//     Term 38 (AT2200-0500)/CC Inputs/Current actual value Ch.30 <-> Data Pointer/CurrentActualValues[29]
//     Term 38 (AT2200-0500)/CC Inputs/Current actual value Ch.4 <-> Data Pointer/CurrentActualValues[3]
//     Term 38 (AT2200-0500)/CC Inputs/Current actual value Ch.5 <-> Data Pointer/CurrentActualValues[4]
//     Term 38 (AT2200-0500)/CC Inputs/Current actual value Ch.6 <-> Data Pointer/CurrentActualValues[5]
//     Term 38 (AT2200-0500)/CC Inputs/Current actual value Ch.7 <-> Data Pointer/CurrentActualValues[6]
//     Term 38 (AT2200-0500)/CC Inputs/Current actual value Ch.8 <-> Data Pointer/CurrentActualValues[7]
//     Term 38 (AT2200-0500)/CC Inputs/Current actual value Ch.9 <-> Data Pointer/CurrentActualValues[8]
//     Term 38 (AT2200-0500)/CC Inputs/Status <-> Data Pointer/Status
//     Term 38 (AT2200-0500)/CC Outputs/Control <-> Data Pointer/Control
//     Term 38 (AT2200-0500)/CC Outputs/Current setpoint value Ch.1 <-> Data Pointer/CurrentSetpointValues[0]
//     Term 38 (AT2200-0500)/CC Outputs/Current setpoint value Ch.10 <-> Data Pointer/CurrentSetpointValues[9]
//     Term 38 (AT2200-0500)/CC Outputs/Current setpoint value Ch.11 <-> Data Pointer/CurrentSetpointValues[10]
//     Term 38 (AT2200-0500)/CC Outputs/Current setpoint value Ch.12 <-> Data Pointer/CurrentSetpointValues[11]
//     Term 38 (AT2200-0500)/CC Outputs/Current setpoint value Ch.13 <-> Data Pointer/CurrentSetpointValues[12]
//     Term 38 (AT2200-0500)/CC Outputs/Current setpoint value Ch.14 <-> Data Pointer/CurrentSetpointValues[13]
//     Term 38 (AT2200-0500)/CC Outputs/Current setpoint value Ch.15 <-> Data Pointer/CurrentSetpointValues[14]
//     Term 38 (AT2200-0500)/CC Outputs/Current setpoint value Ch.16 <-> Data Pointer/CurrentSetpointValues[15]
//     Term 38 (AT2200-0500)/CC Outputs/Current setpoint value Ch.17 <-> Data Pointer/CurrentSetpointValues[16]
//     Term 38 (AT2200-0500)/CC Outputs/Current setpoint value Ch.18 <-> Data Pointer/CurrentSetpointValues[17]
//     Term 38 (AT2200-0500)/CC Outputs/Current setpoint value Ch.19 <-> Data Pointer/CurrentSetpointValues[18]
//     Term 38 (AT2200-0500)/CC Outputs/Current setpoint value Ch.2 <-> Data Pointer/CurrentSetpointValues[1]
//     Term 38 (AT2200-0500)/CC Outputs/Current setpoint value Ch.20 <-> Data Pointer/CurrentSetpointValues[19]
//     Term 38 (AT2200-0500)/CC Outputs/Current setpoint value Ch.21 <-> Data Pointer/CurrentSetpointValues[20]
//     Term 38 (AT2200-0500)/CC Outputs/Current setpoint value Ch.22 <-> Data Pointer/CurrentSetpointValues[21]
//     Term 38 (AT2200-0500)/CC Outputs/Current setpoint value Ch.23 <-> Data Pointer/CurrentSetpointValues[22]
//     Term 38 (AT2200-0500)/CC Outputs/Current setpoint value Ch.24 <-> Data Pointer/CurrentSetpointValues[23]
//     Term 38 (AT2200-0500)/CC Outputs/Current setpoint value Ch.25 <-> Data Pointer/CurrentSetpointValues[24]
//     Term 38 (AT2200-0500)/CC Outputs/Current setpoint value Ch.26 <-> Data Pointer/CurrentSetpointValues[25]
//     Term 38 (AT2200-0500)/CC Outputs/Current setpoint value Ch.27 <-> Data Pointer/CurrentSetpointValues[26]
//     Term 38 (AT2200-0500)/CC Outputs/Current setpoint value Ch.28 <-> Data Pointer/CurrentSetpointValues[27]
//     Term 38 (AT2200-0500)/CC Outputs/Current setpoint value Ch.29 <-> Data Pointer/CurrentSetpointValues[28]
//     Term 38 (AT2200-0500)/CC Outputs/Current setpoint value Ch.3 <-> Data Pointer/CurrentSetpointValues[2]
//     Term 38 (AT2200-0500)/CC Outputs/Current setpoint value Ch.30 <-> Data Pointer/CurrentSetpointValues[29]
//     Term 38 (AT2200-0500)/CC Outputs/Current setpoint value Ch.4 <-> Data Pointer/CurrentSetpointValues[3]
//     Term 38 (AT2200-0500)/CC Outputs/Current setpoint value Ch.5 <-> Data Pointer/CurrentSetpointValues[4]
//     Term 38 (AT2200-0500)/CC Outputs/Current setpoint value Ch.6 <-> Data Pointer/CurrentSetpointValues[5]
//     Term 38 (AT2200-0500)/CC Outputs/Current setpoint value Ch.7 <-> Data Pointer/CurrentSetpointValues[6]
//     Term 38 (AT2200-0500)/CC Outputs/Current setpoint value Ch.8 <-> Data Pointer/CurrentSetpointValues[7]
//     Term 38 (AT2200-0500)/CC Outputs/Current setpoint value Ch.9 <-> Data Pointer/CurrentSetpointValues[8]
//     Term 38 (AT2200-0500)/LFB Inputs/BinaryData <-> Data Pointer/HallSensorValues
//   Device 25 <-> TcCOM Objects/XTS ProcessingUnit 1/Part 1/Module 31
//     Term 39 (AT2000-0250)/CC Inputs/Current actual value Ch.1 <-> Data Pointer/CurrentActualValues[0]
//     Term 39 (AT2000-0250)/CC Inputs/Current actual value Ch.10 <-> Data Pointer/CurrentActualValues[9]
//     Term 39 (AT2000-0250)/CC Inputs/Current actual value Ch.11 <-> Data Pointer/CurrentActualValues[10]
//     Term 39 (AT2000-0250)/CC Inputs/Current actual value Ch.12 <-> Data Pointer/CurrentActualValues[11]
//     Term 39 (AT2000-0250)/CC Inputs/Current actual value Ch.13 <-> Data Pointer/CurrentActualValues[12]
//     Term 39 (AT2000-0250)/CC Inputs/Current actual value Ch.14 <-> Data Pointer/CurrentActualValues[13]
//     Term 39 (AT2000-0250)/CC Inputs/Current actual value Ch.15 <-> Data Pointer/CurrentActualValues[14]
//     Term 39 (AT2000-0250)/CC Inputs/Current actual value Ch.2 <-> Data Pointer/CurrentActualValues[1]
//     Term 39 (AT2000-0250)/CC Inputs/Current actual value Ch.3 <-> Data Pointer/CurrentActualValues[2]
//     Term 39 (AT2000-0250)/CC Inputs/Current actual value Ch.4 <-> Data Pointer/CurrentActualValues[3]
//     Term 39 (AT2000-0250)/CC Inputs/Current actual value Ch.5 <-> Data Pointer/CurrentActualValues[4]
//     Term 39 (AT2000-0250)/CC Inputs/Current actual value Ch.6 <-> Data Pointer/CurrentActualValues[5]
//     Term 39 (AT2000-0250)/CC Inputs/Current actual value Ch.7 <-> Data Pointer/CurrentActualValues[6]
//     Term 39 (AT2000-0250)/CC Inputs/Current actual value Ch.8 <-> Data Pointer/CurrentActualValues[7]
//     Term 39 (AT2000-0250)/CC Inputs/Current actual value Ch.9 <-> Data Pointer/CurrentActualValues[8]
//     Term 39 (AT2000-0250)/CC Inputs/Status <-> Data Pointer/Status
//     Term 39 (AT2000-0250)/CC Outputs/Control <-> Data Pointer/Control
//     Term 39 (AT2000-0250)/CC Outputs/Current setpoint value Ch.1 <-> Data Pointer/CurrentSetpointValues[0]
//     Term 39 (AT2000-0250)/CC Outputs/Current setpoint value Ch.10 <-> Data Pointer/CurrentSetpointValues[9]
//     Term 39 (AT2000-0250)/CC Outputs/Current setpoint value Ch.11 <-> Data Pointer/CurrentSetpointValues[10]
//     Term 39 (AT2000-0250)/CC Outputs/Current setpoint value Ch.12 <-> Data Pointer/CurrentSetpointValues[11]
//     Term 39 (AT2000-0250)/CC Outputs/Current setpoint value Ch.13 <-> Data Pointer/CurrentSetpointValues[12]
//     Term 39 (AT2000-0250)/CC Outputs/Current setpoint value Ch.14 <-> Data Pointer/CurrentSetpointValues[13]
//     Term 39 (AT2000-0250)/CC Outputs/Current setpoint value Ch.15 <-> Data Pointer/CurrentSetpointValues[14]
//     Term 39 (AT2000-0250)/CC Outputs/Current setpoint value Ch.2 <-> Data Pointer/CurrentSetpointValues[1]
//     Term 39 (AT2000-0250)/CC Outputs/Current setpoint value Ch.3 <-> Data Pointer/CurrentSetpointValues[2]
//     Term 39 (AT2000-0250)/CC Outputs/Current setpoint value Ch.4 <-> Data Pointer/CurrentSetpointValues[3]
//     Term 39 (AT2000-0250)/CC Outputs/Current setpoint value Ch.5 <-> Data Pointer/CurrentSetpointValues[4]
//     Term 39 (AT2000-0250)/CC Outputs/Current setpoint value Ch.6 <-> Data Pointer/CurrentSetpointValues[5]
//     Term 39 (AT2000-0250)/CC Outputs/Current setpoint value Ch.7 <-> Data Pointer/CurrentSetpointValues[6]
//     Term 39 (AT2000-0250)/CC Outputs/Current setpoint value Ch.8 <-> Data Pointer/CurrentSetpointValues[7]
//     Term 39 (AT2000-0250)/CC Outputs/Current setpoint value Ch.9 <-> Data Pointer/CurrentSetpointValues[8]
//     Term 39 (AT2000-0250)/Term 40 (AT2000-5250)/FB Inputs/Value Channel 01 <-> Data Pointer/RawPositionValues[0]
//     Term 39 (AT2000-0250)/Term 40 (AT2000-5250)/FB Inputs/Value Channel 02 <-> Data Pointer/RawPositionValues[1]
//     Term 39 (AT2000-0250)/Term 40 (AT2000-5250)/FB Inputs/Value Channel 03 <-> Data Pointer/RawPositionValues[2]
//     Term 39 (AT2000-0250)/Term 40 (AT2000-5250)/FB Inputs/Value Channel 04 <-> Data Pointer/RawPositionValues[3]
//     Term 39 (AT2000-0250)/Term 40 (AT2000-5250)/FB Inputs/Value Channel 05 <-> Data Pointer/RawPositionValues[4]
//     Term 39 (AT2000-0250)/Term 40 (AT2000-5250)/FB Inputs/Value Channel 06 <-> Data Pointer/RawPositionValues[5]
//     Term 39 (AT2000-0250)/Term 40 (AT2000-5250)/FB Inputs/Value Channel 07 <-> Data Pointer/RawPositionValues[6]
//     Term 39 (AT2000-0250)/Term 40 (AT2000-5250)/FB Inputs/Value Channel 08 <-> Data Pointer/RawPositionValues[7]
//     Term 39 (AT2000-0250)/Term 40 (AT2000-5250)/FB Inputs/Value Channel 09 <-> Data Pointer/RawPositionValues[8]
//     Term 39 (AT2000-0250)/Term 40 (AT2000-5250)/FB Inputs/Value Channel 10 <-> Data Pointer/RawPositionValues[9]
//     Term 39 (AT2000-0250)/Term 40 (AT2000-5250)/FB Inputs/Value Channel 11 <-> Data Pointer/RawPositionValues[10]
//     Term 39 (AT2000-0250)/Term 40 (AT2000-5250)/FB Inputs/Value Channel 12 <-> Data Pointer/RawPositionValues[11]
//     Term 39 (AT2000-0250)/Term 40 (AT2000-5250)/FB Inputs/Value Channel 13 <-> Data Pointer/RawPositionValues[12]
//     Term 39 (AT2000-0250)/Term 40 (AT2000-5250)/FB Inputs/Value Channel 14 <-> Data Pointer/RawPositionValues[13]
//     Term 39 (AT2000-0250)/Term 40 (AT2000-5250)/FB Inputs/Value Channel 15 <-> Data Pointer/RawPositionValues[14]
//     Term 39 (AT2000-0250)/Term 40 (AT2000-5250)/FB Inputs/Value Channel 16 <-> Data Pointer/RawPositionValues[15]
//     Term 39 (AT2000-0250)/Term 40 (AT2000-5250)/FB Inputs/Value Channel 17 <-> Data Pointer/RawPositionValues[16]
//     Term 39 (AT2000-0250)/Term 40 (AT2000-5250)/FB Inputs/Value Channel 18 <-> Data Pointer/RawPositionValues[17]
//     Term 39 (AT2000-0250)/Term 40 (AT2000-5250)/FB Inputs/Value Channel 19 <-> Data Pointer/RawPositionValues[18]
//     Term 39 (AT2000-0250)/Term 40 (AT2000-5250)/FB Inputs/Value Channel 20 <-> Data Pointer/RawPositionValues[19]
//     Term 39 (AT2000-0250)/Term 40 (AT2000-5250)/FB Inputs/Value Channel 21 <-> Data Pointer/RawPositionValues[20]
//     Term 39 (AT2000-0250)/Term 40 (AT2000-5250)/FB Inputs/Value Channel 22 <-> Data Pointer/RawPositionValues[21]
//     Term 39 (AT2000-0250)/Term 40 (AT2000-5250)/FB Inputs/Value Channel 23 <-> Data Pointer/RawPositionValues[22]
//     Term 39 (AT2000-0250)/Term 40 (AT2000-5250)/FB Inputs/Value Channel 24 <-> Data Pointer/RawPositionValues[23]
//     Term 39 (AT2000-0250)/Term 40 (AT2000-5250)/FB Inputs/Value Channel 25 <-> Data Pointer/RawPositionValues[24]
//     Term 39 (AT2000-0250)/Term 40 (AT2000-5250)/FB Inputs/Value Channel 26 <-> Data Pointer/RawPositionValues[25]
//     Term 39 (AT2000-0250)/Term 40 (AT2000-5250)/FB Inputs/Value Channel 27 <-> Data Pointer/RawPositionValues[26]
//     Term 39 (AT2000-0250)/Term 40 (AT2000-5250)/FB Inputs/Value Channel 28 <-> Data Pointer/RawPositionValues[27]
//     Term 39 (AT2000-0250)/Term 40 (AT2000-5250)/FB Inputs/Value Channel 29 <-> Data Pointer/RawPositionValues[28]
//     Term 39 (AT2000-0250)/Term 40 (AT2000-5250)/FB Inputs/Value Channel 30 <-> Data Pointer/RawPositionValues[29]
//     Term 39 (AT2000-0250)/Term 40 (AT2000-5250)/FB Inputs/Value Channel 31 <-> Data Pointer/RawPositionValues[30]
//     Term 39 (AT2000-0250)/Term 40 (AT2000-5250)/FB Inputs/Value Channel 32 <-> Data Pointer/RawPositionValues[31]
//   Device 26 <-> TcCOM Objects/XTS ProcessingUnit 1/Part 1/Module 32
//     Term 41 (AT2002-0250)/CC Inputs/Current actual value Ch.1 <-> Data Pointer/CurrentActualValues[0]
//     Term 41 (AT2002-0250)/CC Inputs/Current actual value Ch.10 <-> Data Pointer/CurrentActualValues[9]
//     Term 41 (AT2002-0250)/CC Inputs/Current actual value Ch.11 <-> Data Pointer/CurrentActualValues[10]
//     Term 41 (AT2002-0250)/CC Inputs/Current actual value Ch.12 <-> Data Pointer/CurrentActualValues[11]
//     Term 41 (AT2002-0250)/CC Inputs/Current actual value Ch.13 <-> Data Pointer/CurrentActualValues[12]
//     Term 41 (AT2002-0250)/CC Inputs/Current actual value Ch.14 <-> Data Pointer/CurrentActualValues[13]
//     Term 41 (AT2002-0250)/CC Inputs/Current actual value Ch.15 <-> Data Pointer/CurrentActualValues[14]
//     Term 41 (AT2002-0250)/CC Inputs/Current actual value Ch.2 <-> Data Pointer/CurrentActualValues[1]
//     Term 41 (AT2002-0250)/CC Inputs/Current actual value Ch.3 <-> Data Pointer/CurrentActualValues[2]
//     Term 41 (AT2002-0250)/CC Inputs/Current actual value Ch.4 <-> Data Pointer/CurrentActualValues[3]
//     Term 41 (AT2002-0250)/CC Inputs/Current actual value Ch.5 <-> Data Pointer/CurrentActualValues[4]
//     Term 41 (AT2002-0250)/CC Inputs/Current actual value Ch.6 <-> Data Pointer/CurrentActualValues[5]
//     Term 41 (AT2002-0250)/CC Inputs/Current actual value Ch.7 <-> Data Pointer/CurrentActualValues[6]
//     Term 41 (AT2002-0250)/CC Inputs/Current actual value Ch.8 <-> Data Pointer/CurrentActualValues[7]
//     Term 41 (AT2002-0250)/CC Inputs/Current actual value Ch.9 <-> Data Pointer/CurrentActualValues[8]
//     Term 41 (AT2002-0250)/CC Inputs/Status <-> Data Pointer/Status
//     Term 41 (AT2002-0250)/CC Outputs/Control <-> Data Pointer/Control
//     Term 41 (AT2002-0250)/CC Outputs/Current setpoint value Ch.1 <-> Data Pointer/CurrentSetpointValues[0]
//     Term 41 (AT2002-0250)/CC Outputs/Current setpoint value Ch.10 <-> Data Pointer/CurrentSetpointValues[9]
//     Term 41 (AT2002-0250)/CC Outputs/Current setpoint value Ch.11 <-> Data Pointer/CurrentSetpointValues[10]
//     Term 41 (AT2002-0250)/CC Outputs/Current setpoint value Ch.12 <-> Data Pointer/CurrentSetpointValues[11]
//     Term 41 (AT2002-0250)/CC Outputs/Current setpoint value Ch.13 <-> Data Pointer/CurrentSetpointValues[12]
//     Term 41 (AT2002-0250)/CC Outputs/Current setpoint value Ch.14 <-> Data Pointer/CurrentSetpointValues[13]
//     Term 41 (AT2002-0250)/CC Outputs/Current setpoint value Ch.15 <-> Data Pointer/CurrentSetpointValues[14]
//     Term 41 (AT2002-0250)/CC Outputs/Current setpoint value Ch.2 <-> Data Pointer/CurrentSetpointValues[1]
//     Term 41 (AT2002-0250)/CC Outputs/Current setpoint value Ch.3 <-> Data Pointer/CurrentSetpointValues[2]
//     Term 41 (AT2002-0250)/CC Outputs/Current setpoint value Ch.4 <-> Data Pointer/CurrentSetpointValues[3]
//     Term 41 (AT2002-0250)/CC Outputs/Current setpoint value Ch.5 <-> Data Pointer/CurrentSetpointValues[4]
//     Term 41 (AT2002-0250)/CC Outputs/Current setpoint value Ch.6 <-> Data Pointer/CurrentSetpointValues[5]
//     Term 41 (AT2002-0250)/CC Outputs/Current setpoint value Ch.7 <-> Data Pointer/CurrentSetpointValues[6]
//     Term 41 (AT2002-0250)/CC Outputs/Current setpoint value Ch.8 <-> Data Pointer/CurrentSetpointValues[7]
//     Term 41 (AT2002-0250)/CC Outputs/Current setpoint value Ch.9 <-> Data Pointer/CurrentSetpointValues[8]
//     Term 41 (AT2002-0250)/Term 42 (AT2002-5250)/FB Inputs/Value Channel 01 <-> Data Pointer/RawPositionValues[0]
//     Term 41 (AT2002-0250)/Term 42 (AT2002-5250)/FB Inputs/Value Channel 02 <-> Data Pointer/RawPositionValues[1]
//     Term 41 (AT2002-0250)/Term 42 (AT2002-5250)/FB Inputs/Value Channel 03 <-> Data Pointer/RawPositionValues[2]
//     Term 41 (AT2002-0250)/Term 42 (AT2002-5250)/FB Inputs/Value Channel 04 <-> Data Pointer/RawPositionValues[3]
//     Term 41 (AT2002-0250)/Term 42 (AT2002-5250)/FB Inputs/Value Channel 05 <-> Data Pointer/RawPositionValues[4]
//     Term 41 (AT2002-0250)/Term 42 (AT2002-5250)/FB Inputs/Value Channel 06 <-> Data Pointer/RawPositionValues[5]
//     Term 41 (AT2002-0250)/Term 42 (AT2002-5250)/FB Inputs/Value Channel 07 <-> Data Pointer/RawPositionValues[6]
//     Term 41 (AT2002-0250)/Term 42 (AT2002-5250)/FB Inputs/Value Channel 08 <-> Data Pointer/RawPositionValues[7]
//     Term 41 (AT2002-0250)/Term 42 (AT2002-5250)/FB Inputs/Value Channel 09 <-> Data Pointer/RawPositionValues[8]
//     Term 41 (AT2002-0250)/Term 42 (AT2002-5250)/FB Inputs/Value Channel 10 <-> Data Pointer/RawPositionValues[9]
//     Term 41 (AT2002-0250)/Term 42 (AT2002-5250)/FB Inputs/Value Channel 11 <-> Data Pointer/RawPositionValues[10]
//     Term 41 (AT2002-0250)/Term 42 (AT2002-5250)/FB Inputs/Value Channel 12 <-> Data Pointer/RawPositionValues[11]
//     Term 41 (AT2002-0250)/Term 42 (AT2002-5250)/FB Inputs/Value Channel 13 <-> Data Pointer/RawPositionValues[12]
//     Term 41 (AT2002-0250)/Term 42 (AT2002-5250)/FB Inputs/Value Channel 14 <-> Data Pointer/RawPositionValues[13]
//     Term 41 (AT2002-0250)/Term 42 (AT2002-5250)/FB Inputs/Value Channel 15 <-> Data Pointer/RawPositionValues[14]
//     Term 41 (AT2002-0250)/Term 42 (AT2002-5250)/FB Inputs/Value Channel 16 <-> Data Pointer/RawPositionValues[15]
//     Term 41 (AT2002-0250)/Term 42 (AT2002-5250)/FB Inputs/Value Channel 17 <-> Data Pointer/RawPositionValues[16]
//     Term 41 (AT2002-0250)/Term 42 (AT2002-5250)/FB Inputs/Value Channel 18 <-> Data Pointer/RawPositionValues[17]
//     Term 41 (AT2002-0250)/Term 42 (AT2002-5250)/FB Inputs/Value Channel 19 <-> Data Pointer/RawPositionValues[18]
//     Term 41 (AT2002-0250)/Term 42 (AT2002-5250)/FB Inputs/Value Channel 20 <-> Data Pointer/RawPositionValues[19]
//     Term 41 (AT2002-0250)/Term 42 (AT2002-5250)/FB Inputs/Value Channel 21 <-> Data Pointer/RawPositionValues[20]
//     Term 41 (AT2002-0250)/Term 42 (AT2002-5250)/FB Inputs/Value Channel 22 <-> Data Pointer/RawPositionValues[21]
//     Term 41 (AT2002-0250)/Term 42 (AT2002-5250)/FB Inputs/Value Channel 23 <-> Data Pointer/RawPositionValues[22]
//     Term 41 (AT2002-0250)/Term 42 (AT2002-5250)/FB Inputs/Value Channel 24 <-> Data Pointer/RawPositionValues[23]
//     Term 41 (AT2002-0250)/Term 42 (AT2002-5250)/FB Inputs/Value Channel 25 <-> Data Pointer/RawPositionValues[24]
//     Term 41 (AT2002-0250)/Term 42 (AT2002-5250)/FB Inputs/Value Channel 26 <-> Data Pointer/RawPositionValues[25]
//     Term 41 (AT2002-0250)/Term 42 (AT2002-5250)/FB Inputs/Value Channel 27 <-> Data Pointer/RawPositionValues[26]
//     Term 41 (AT2002-0250)/Term 42 (AT2002-5250)/FB Inputs/Value Channel 28 <-> Data Pointer/RawPositionValues[27]
//     Term 41 (AT2002-0250)/Term 42 (AT2002-5250)/FB Inputs/Value Channel 29 <-> Data Pointer/RawPositionValues[28]
//     Term 41 (AT2002-0250)/Term 42 (AT2002-5250)/FB Inputs/Value Channel 30 <-> Data Pointer/RawPositionValues[29]
//     Term 41 (AT2002-0250)/Term 42 (AT2002-5250)/FB Inputs/Value Channel 31 <-> Data Pointer/RawPositionValues[30]
//     Term 41 (AT2002-0250)/Term 42 (AT2002-5250)/FB Inputs/Value Channel 32 <-> Data Pointer/RawPositionValues[31]
//   Device 26 <-> TcCOM Objects/XTS ProcessingUnit 1/Part 1/Module 33
//     Term 43 (AT2200-0500)/CC Inputs/Current actual value Ch.1 <-> Data Pointer/CurrentActualValues[0]
//     Term 43 (AT2200-0500)/CC Inputs/Current actual value Ch.10 <-> Data Pointer/CurrentActualValues[9]
//     Term 43 (AT2200-0500)/CC Inputs/Current actual value Ch.11 <-> Data Pointer/CurrentActualValues[10]
//     Term 43 (AT2200-0500)/CC Inputs/Current actual value Ch.12 <-> Data Pointer/CurrentActualValues[11]
//     Term 43 (AT2200-0500)/CC Inputs/Current actual value Ch.13 <-> Data Pointer/CurrentActualValues[12]
//     Term 43 (AT2200-0500)/CC Inputs/Current actual value Ch.14 <-> Data Pointer/CurrentActualValues[13]
//     Term 43 (AT2200-0500)/CC Inputs/Current actual value Ch.15 <-> Data Pointer/CurrentActualValues[14]
//     Term 43 (AT2200-0500)/CC Inputs/Current actual value Ch.16 <-> Data Pointer/CurrentActualValues[15]
//     Term 43 (AT2200-0500)/CC Inputs/Current actual value Ch.17 <-> Data Pointer/CurrentActualValues[16]
//     Term 43 (AT2200-0500)/CC Inputs/Current actual value Ch.18 <-> Data Pointer/CurrentActualValues[17]
//     Term 43 (AT2200-0500)/CC Inputs/Current actual value Ch.19 <-> Data Pointer/CurrentActualValues[18]
//     Term 43 (AT2200-0500)/CC Inputs/Current actual value Ch.2 <-> Data Pointer/CurrentActualValues[1]
//     Term 43 (AT2200-0500)/CC Inputs/Current actual value Ch.20 <-> Data Pointer/CurrentActualValues[19]
//     Term 43 (AT2200-0500)/CC Inputs/Current actual value Ch.21 <-> Data Pointer/CurrentActualValues[20]
//     Term 43 (AT2200-0500)/CC Inputs/Current actual value Ch.22 <-> Data Pointer/CurrentActualValues[21]
//     Term 43 (AT2200-0500)/CC Inputs/Current actual value Ch.23 <-> Data Pointer/CurrentActualValues[22]
//     Term 43 (AT2200-0500)/CC Inputs/Current actual value Ch.24 <-> Data Pointer/CurrentActualValues[23]
//     Term 43 (AT2200-0500)/CC Inputs/Current actual value Ch.25 <-> Data Pointer/CurrentActualValues[24]
//     Term 43 (AT2200-0500)/CC Inputs/Current actual value Ch.26 <-> Data Pointer/CurrentActualValues[25]
//     Term 43 (AT2200-0500)/CC Inputs/Current actual value Ch.27 <-> Data Pointer/CurrentActualValues[26]
//     Term 43 (AT2200-0500)/CC Inputs/Current actual value Ch.28 <-> Data Pointer/CurrentActualValues[27]
//     Term 43 (AT2200-0500)/CC Inputs/Current actual value Ch.29 <-> Data Pointer/CurrentActualValues[28]
//     Term 43 (AT2200-0500)/CC Inputs/Current actual value Ch.3 <-> Data Pointer/CurrentActualValues[2]
//     Term 43 (AT2200-0500)/CC Inputs/Current actual value Ch.30 <-> Data Pointer/CurrentActualValues[29]
//     Term 43 (AT2200-0500)/CC Inputs/Current actual value Ch.4 <-> Data Pointer/CurrentActualValues[3]
//     Term 43 (AT2200-0500)/CC Inputs/Current actual value Ch.5 <-> Data Pointer/CurrentActualValues[4]
//     Term 43 (AT2200-0500)/CC Inputs/Current actual value Ch.6 <-> Data Pointer/CurrentActualValues[5]
//     Term 43 (AT2200-0500)/CC Inputs/Current actual value Ch.7 <-> Data Pointer/CurrentActualValues[6]
//     Term 43 (AT2200-0500)/CC Inputs/Current actual value Ch.8 <-> Data Pointer/CurrentActualValues[7]
//     Term 43 (AT2200-0500)/CC Inputs/Current actual value Ch.9 <-> Data Pointer/CurrentActualValues[8]
//     Term 43 (AT2200-0500)/CC Inputs/Status <-> Data Pointer/Status
//     Term 43 (AT2200-0500)/CC Outputs/Control <-> Data Pointer/Control
//     Term 43 (AT2200-0500)/CC Outputs/Current setpoint value Ch.1 <-> Data Pointer/CurrentSetpointValues[0]
//     Term 43 (AT2200-0500)/CC Outputs/Current setpoint value Ch.10 <-> Data Pointer/CurrentSetpointValues[9]
//     Term 43 (AT2200-0500)/CC Outputs/Current setpoint value Ch.11 <-> Data Pointer/CurrentSetpointValues[10]
//     Term 43 (AT2200-0500)/CC Outputs/Current setpoint value Ch.12 <-> Data Pointer/CurrentSetpointValues[11]
//     Term 43 (AT2200-0500)/CC Outputs/Current setpoint value Ch.13 <-> Data Pointer/CurrentSetpointValues[12]
//     Term 43 (AT2200-0500)/CC Outputs/Current setpoint value Ch.14 <-> Data Pointer/CurrentSetpointValues[13]
//     Term 43 (AT2200-0500)/CC Outputs/Current setpoint value Ch.15 <-> Data Pointer/CurrentSetpointValues[14]
//     Term 43 (AT2200-0500)/CC Outputs/Current setpoint value Ch.16 <-> Data Pointer/CurrentSetpointValues[15]
//     Term 43 (AT2200-0500)/CC Outputs/Current setpoint value Ch.17 <-> Data Pointer/CurrentSetpointValues[16]
//     Term 43 (AT2200-0500)/CC Outputs/Current setpoint value Ch.18 <-> Data Pointer/CurrentSetpointValues[17]
//     Term 43 (AT2200-0500)/CC Outputs/Current setpoint value Ch.19 <-> Data Pointer/CurrentSetpointValues[18]
//     Term 43 (AT2200-0500)/CC Outputs/Current setpoint value Ch.2 <-> Data Pointer/CurrentSetpointValues[1]
//     Term 43 (AT2200-0500)/CC Outputs/Current setpoint value Ch.20 <-> Data Pointer/CurrentSetpointValues[19]
//     Term 43 (AT2200-0500)/CC Outputs/Current setpoint value Ch.21 <-> Data Pointer/CurrentSetpointValues[20]
//     Term 43 (AT2200-0500)/CC Outputs/Current setpoint value Ch.22 <-> Data Pointer/CurrentSetpointValues[21]
//     Term 43 (AT2200-0500)/CC Outputs/Current setpoint value Ch.23 <-> Data Pointer/CurrentSetpointValues[22]
//     Term 43 (AT2200-0500)/CC Outputs/Current setpoint value Ch.24 <-> Data Pointer/CurrentSetpointValues[23]
//     Term 43 (AT2200-0500)/CC Outputs/Current setpoint value Ch.25 <-> Data Pointer/CurrentSetpointValues[24]
//     Term 43 (AT2200-0500)/CC Outputs/Current setpoint value Ch.26 <-> Data Pointer/CurrentSetpointValues[25]
//     Term 43 (AT2200-0500)/CC Outputs/Current setpoint value Ch.27 <-> Data Pointer/CurrentSetpointValues[26]
//     Term 43 (AT2200-0500)/CC Outputs/Current setpoint value Ch.28 <-> Data Pointer/CurrentSetpointValues[27]
//     Term 43 (AT2200-0500)/CC Outputs/Current setpoint value Ch.29 <-> Data Pointer/CurrentSetpointValues[28]
//     Term 43 (AT2200-0500)/CC Outputs/Current setpoint value Ch.3 <-> Data Pointer/CurrentSetpointValues[2]
//     Term 43 (AT2200-0500)/CC Outputs/Current setpoint value Ch.30 <-> Data Pointer/CurrentSetpointValues[29]
//     Term 43 (AT2200-0500)/CC Outputs/Current setpoint value Ch.4 <-> Data Pointer/CurrentSetpointValues[3]
//     Term 43 (AT2200-0500)/CC Outputs/Current setpoint value Ch.5 <-> Data Pointer/CurrentSetpointValues[4]
//     Term 43 (AT2200-0500)/CC Outputs/Current setpoint value Ch.6 <-> Data Pointer/CurrentSetpointValues[5]
//     Term 43 (AT2200-0500)/CC Outputs/Current setpoint value Ch.7 <-> Data Pointer/CurrentSetpointValues[6]
//     Term 43 (AT2200-0500)/CC Outputs/Current setpoint value Ch.8 <-> Data Pointer/CurrentSetpointValues[7]
//     Term 43 (AT2200-0500)/CC Outputs/Current setpoint value Ch.9 <-> Data Pointer/CurrentSetpointValues[8]
//     Term 43 (AT2200-0500)/LFB Inputs/BinaryData <-> Data Pointer/HallSensorValues
//   Device 26 <-> TcCOM Objects/XTS ProcessingUnit 1/Part 1/Module 34
//     Term 44 (AT2200-0500)/CC Inputs/Current actual value Ch.1 <-> Data Pointer/CurrentActualValues[0]
//     Term 44 (AT2200-0500)/CC Inputs/Current actual value Ch.10 <-> Data Pointer/CurrentActualValues[9]
//     Term 44 (AT2200-0500)/CC Inputs/Current actual value Ch.11 <-> Data Pointer/CurrentActualValues[10]
//     Term 44 (AT2200-0500)/CC Inputs/Current actual value Ch.12 <-> Data Pointer/CurrentActualValues[11]
//     Term 44 (AT2200-0500)/CC Inputs/Current actual value Ch.13 <-> Data Pointer/CurrentActualValues[12]
//     Term 44 (AT2200-0500)/CC Inputs/Current actual value Ch.14 <-> Data Pointer/CurrentActualValues[13]
//     Term 44 (AT2200-0500)/CC Inputs/Current actual value Ch.15 <-> Data Pointer/CurrentActualValues[14]
//     Term 44 (AT2200-0500)/CC Inputs/Current actual value Ch.16 <-> Data Pointer/CurrentActualValues[15]
//     Term 44 (AT2200-0500)/CC Inputs/Current actual value Ch.17 <-> Data Pointer/CurrentActualValues[16]
//     Term 44 (AT2200-0500)/CC Inputs/Current actual value Ch.18 <-> Data Pointer/CurrentActualValues[17]
//     Term 44 (AT2200-0500)/CC Inputs/Current actual value Ch.19 <-> Data Pointer/CurrentActualValues[18]
//     Term 44 (AT2200-0500)/CC Inputs/Current actual value Ch.2 <-> Data Pointer/CurrentActualValues[1]
//     Term 44 (AT2200-0500)/CC Inputs/Current actual value Ch.20 <-> Data Pointer/CurrentActualValues[19]
//     Term 44 (AT2200-0500)/CC Inputs/Current actual value Ch.21 <-> Data Pointer/CurrentActualValues[20]
//     Term 44 (AT2200-0500)/CC Inputs/Current actual value Ch.22 <-> Data Pointer/CurrentActualValues[21]
//     Term 44 (AT2200-0500)/CC Inputs/Current actual value Ch.23 <-> Data Pointer/CurrentActualValues[22]
//     Term 44 (AT2200-0500)/CC Inputs/Current actual value Ch.24 <-> Data Pointer/CurrentActualValues[23]
//     Term 44 (AT2200-0500)/CC Inputs/Current actual value Ch.25 <-> Data Pointer/CurrentActualValues[24]
//     Term 44 (AT2200-0500)/CC Inputs/Current actual value Ch.26 <-> Data Pointer/CurrentActualValues[25]
//     Term 44 (AT2200-0500)/CC Inputs/Current actual value Ch.27 <-> Data Pointer/CurrentActualValues[26]
//     Term 44 (AT2200-0500)/CC Inputs/Current actual value Ch.28 <-> Data Pointer/CurrentActualValues[27]
//     Term 44 (AT2200-0500)/CC Inputs/Current actual value Ch.29 <-> Data Pointer/CurrentActualValues[28]
//     Term 44 (AT2200-0500)/CC Inputs/Current actual value Ch.3 <-> Data Pointer/CurrentActualValues[2]
//     Term 44 (AT2200-0500)/CC Inputs/Current actual value Ch.30 <-> Data Pointer/CurrentActualValues[29]
//     Term 44 (AT2200-0500)/CC Inputs/Current actual value Ch.4 <-> Data Pointer/CurrentActualValues[3]
//     Term 44 (AT2200-0500)/CC Inputs/Current actual value Ch.5 <-> Data Pointer/CurrentActualValues[4]
//     Term 44 (AT2200-0500)/CC Inputs/Current actual value Ch.6 <-> Data Pointer/CurrentActualValues[5]
//     Term 44 (AT2200-0500)/CC Inputs/Current actual value Ch.7 <-> Data Pointer/CurrentActualValues[6]
//     Term 44 (AT2200-0500)/CC Inputs/Current actual value Ch.8 <-> Data Pointer/CurrentActualValues[7]
//     Term 44 (AT2200-0500)/CC Inputs/Current actual value Ch.9 <-> Data Pointer/CurrentActualValues[8]
//     Term 44 (AT2200-0500)/CC Inputs/Status <-> Data Pointer/Status
//     Term 44 (AT2200-0500)/CC Outputs/Control <-> Data Pointer/Control
//     Term 44 (AT2200-0500)/CC Outputs/Current setpoint value Ch.1 <-> Data Pointer/CurrentSetpointValues[0]
//     Term 44 (AT2200-0500)/CC Outputs/Current setpoint value Ch.10 <-> Data Pointer/CurrentSetpointValues[9]
//     Term 44 (AT2200-0500)/CC Outputs/Current setpoint value Ch.11 <-> Data Pointer/CurrentSetpointValues[10]
//     Term 44 (AT2200-0500)/CC Outputs/Current setpoint value Ch.12 <-> Data Pointer/CurrentSetpointValues[11]
//     Term 44 (AT2200-0500)/CC Outputs/Current setpoint value Ch.13 <-> Data Pointer/CurrentSetpointValues[12]
//     Term 44 (AT2200-0500)/CC Outputs/Current setpoint value Ch.14 <-> Data Pointer/CurrentSetpointValues[13]
//     Term 44 (AT2200-0500)/CC Outputs/Current setpoint value Ch.15 <-> Data Pointer/CurrentSetpointValues[14]
//     Term 44 (AT2200-0500)/CC Outputs/Current setpoint value Ch.16 <-> Data Pointer/CurrentSetpointValues[15]
//     Term 44 (AT2200-0500)/CC Outputs/Current setpoint value Ch.17 <-> Data Pointer/CurrentSetpointValues[16]
//     Term 44 (AT2200-0500)/CC Outputs/Current setpoint value Ch.18 <-> Data Pointer/CurrentSetpointValues[17]
//     Term 44 (AT2200-0500)/CC Outputs/Current setpoint value Ch.19 <-> Data Pointer/CurrentSetpointValues[18]
//     Term 44 (AT2200-0500)/CC Outputs/Current setpoint value Ch.2 <-> Data Pointer/CurrentSetpointValues[1]
//     Term 44 (AT2200-0500)/CC Outputs/Current setpoint value Ch.20 <-> Data Pointer/CurrentSetpointValues[19]
//     Term 44 (AT2200-0500)/CC Outputs/Current setpoint value Ch.21 <-> Data Pointer/CurrentSetpointValues[20]
//     Term 44 (AT2200-0500)/CC Outputs/Current setpoint value Ch.22 <-> Data Pointer/CurrentSetpointValues[21]
//     Term 44 (AT2200-0500)/CC Outputs/Current setpoint value Ch.23 <-> Data Pointer/CurrentSetpointValues[22]
//     Term 44 (AT2200-0500)/CC Outputs/Current setpoint value Ch.24 <-> Data Pointer/CurrentSetpointValues[23]
//     Term 44 (AT2200-0500)/CC Outputs/Current setpoint value Ch.25 <-> Data Pointer/CurrentSetpointValues[24]
//     Term 44 (AT2200-0500)/CC Outputs/Current setpoint value Ch.26 <-> Data Pointer/CurrentSetpointValues[25]
//     Term 44 (AT2200-0500)/CC Outputs/Current setpoint value Ch.27 <-> Data Pointer/CurrentSetpointValues[26]
//     Term 44 (AT2200-0500)/CC Outputs/Current setpoint value Ch.28 <-> Data Pointer/CurrentSetpointValues[27]
//     Term 44 (AT2200-0500)/CC Outputs/Current setpoint value Ch.29 <-> Data Pointer/CurrentSetpointValues[28]
//     Term 44 (AT2200-0500)/CC Outputs/Current setpoint value Ch.3 <-> Data Pointer/CurrentSetpointValues[2]
//     Term 44 (AT2200-0500)/CC Outputs/Current setpoint value Ch.30 <-> Data Pointer/CurrentSetpointValues[29]
//     Term 44 (AT2200-0500)/CC Outputs/Current setpoint value Ch.4 <-> Data Pointer/CurrentSetpointValues[3]
//     Term 44 (AT2200-0500)/CC Outputs/Current setpoint value Ch.5 <-> Data Pointer/CurrentSetpointValues[4]
//     Term 44 (AT2200-0500)/CC Outputs/Current setpoint value Ch.6 <-> Data Pointer/CurrentSetpointValues[5]
//     Term 44 (AT2200-0500)/CC Outputs/Current setpoint value Ch.7 <-> Data Pointer/CurrentSetpointValues[6]
//     Term 44 (AT2200-0500)/CC Outputs/Current setpoint value Ch.8 <-> Data Pointer/CurrentSetpointValues[7]
//     Term 44 (AT2200-0500)/CC Outputs/Current setpoint value Ch.9 <-> Data Pointer/CurrentSetpointValues[8]
//     Term 44 (AT2200-0500)/LFB Inputs/BinaryData <-> Data Pointer/HallSensorValues
//   Device 27 <-> TcCOM Objects/XTS ProcessingUnit 1/Part 1/Module 35
//     Term 45 (AT2202-0500)/CC Inputs/Current actual value Ch.1 <-> Data Pointer/CurrentActualValues[0]
//     Term 45 (AT2202-0500)/CC Inputs/Current actual value Ch.10 <-> Data Pointer/CurrentActualValues[9]
//     Term 45 (AT2202-0500)/CC Inputs/Current actual value Ch.11 <-> Data Pointer/CurrentActualValues[10]
//     Term 45 (AT2202-0500)/CC Inputs/Current actual value Ch.12 <-> Data Pointer/CurrentActualValues[11]
//     Term 45 (AT2202-0500)/CC Inputs/Current actual value Ch.13 <-> Data Pointer/CurrentActualValues[12]
//     Term 45 (AT2202-0500)/CC Inputs/Current actual value Ch.14 <-> Data Pointer/CurrentActualValues[13]
//     Term 45 (AT2202-0500)/CC Inputs/Current actual value Ch.15 <-> Data Pointer/CurrentActualValues[14]
//     Term 45 (AT2202-0500)/CC Inputs/Current actual value Ch.16 <-> Data Pointer/CurrentActualValues[15]
//     Term 45 (AT2202-0500)/CC Inputs/Current actual value Ch.17 <-> Data Pointer/CurrentActualValues[16]
//     Term 45 (AT2202-0500)/CC Inputs/Current actual value Ch.18 <-> Data Pointer/CurrentActualValues[17]
//     Term 45 (AT2202-0500)/CC Inputs/Current actual value Ch.19 <-> Data Pointer/CurrentActualValues[18]
//     Term 45 (AT2202-0500)/CC Inputs/Current actual value Ch.2 <-> Data Pointer/CurrentActualValues[1]
//     Term 45 (AT2202-0500)/CC Inputs/Current actual value Ch.20 <-> Data Pointer/CurrentActualValues[19]
//     Term 45 (AT2202-0500)/CC Inputs/Current actual value Ch.21 <-> Data Pointer/CurrentActualValues[20]
//     Term 45 (AT2202-0500)/CC Inputs/Current actual value Ch.22 <-> Data Pointer/CurrentActualValues[21]
//     Term 45 (AT2202-0500)/CC Inputs/Current actual value Ch.23 <-> Data Pointer/CurrentActualValues[22]
//     Term 45 (AT2202-0500)/CC Inputs/Current actual value Ch.24 <-> Data Pointer/CurrentActualValues[23]
//     Term 45 (AT2202-0500)/CC Inputs/Current actual value Ch.25 <-> Data Pointer/CurrentActualValues[24]
//     Term 45 (AT2202-0500)/CC Inputs/Current actual value Ch.26 <-> Data Pointer/CurrentActualValues[25]
//     Term 45 (AT2202-0500)/CC Inputs/Current actual value Ch.27 <-> Data Pointer/CurrentActualValues[26]
//     Term 45 (AT2202-0500)/CC Inputs/Current actual value Ch.28 <-> Data Pointer/CurrentActualValues[27]
//     Term 45 (AT2202-0500)/CC Inputs/Current actual value Ch.29 <-> Data Pointer/CurrentActualValues[28]
//     Term 45 (AT2202-0500)/CC Inputs/Current actual value Ch.3 <-> Data Pointer/CurrentActualValues[2]
//     Term 45 (AT2202-0500)/CC Inputs/Current actual value Ch.30 <-> Data Pointer/CurrentActualValues[29]
//     Term 45 (AT2202-0500)/CC Inputs/Current actual value Ch.4 <-> Data Pointer/CurrentActualValues[3]
//     Term 45 (AT2202-0500)/CC Inputs/Current actual value Ch.5 <-> Data Pointer/CurrentActualValues[4]
//     Term 45 (AT2202-0500)/CC Inputs/Current actual value Ch.6 <-> Data Pointer/CurrentActualValues[5]
//     Term 45 (AT2202-0500)/CC Inputs/Current actual value Ch.7 <-> Data Pointer/CurrentActualValues[6]
//     Term 45 (AT2202-0500)/CC Inputs/Current actual value Ch.8 <-> Data Pointer/CurrentActualValues[7]
//     Term 45 (AT2202-0500)/CC Inputs/Current actual value Ch.9 <-> Data Pointer/CurrentActualValues[8]
//     Term 45 (AT2202-0500)/CC Inputs/Status <-> Data Pointer/Status
//     Term 45 (AT2202-0500)/CC Outputs/Control <-> Data Pointer/Control
//     Term 45 (AT2202-0500)/CC Outputs/Current setpoint value Ch.1 <-> Data Pointer/CurrentSetpointValues[0]
//     Term 45 (AT2202-0500)/CC Outputs/Current setpoint value Ch.10 <-> Data Pointer/CurrentSetpointValues[9]
//     Term 45 (AT2202-0500)/CC Outputs/Current setpoint value Ch.11 <-> Data Pointer/CurrentSetpointValues[10]
//     Term 45 (AT2202-0500)/CC Outputs/Current setpoint value Ch.12 <-> Data Pointer/CurrentSetpointValues[11]
//     Term 45 (AT2202-0500)/CC Outputs/Current setpoint value Ch.13 <-> Data Pointer/CurrentSetpointValues[12]
//     Term 45 (AT2202-0500)/CC Outputs/Current setpoint value Ch.14 <-> Data Pointer/CurrentSetpointValues[13]
//     Term 45 (AT2202-0500)/CC Outputs/Current setpoint value Ch.15 <-> Data Pointer/CurrentSetpointValues[14]
//     Term 45 (AT2202-0500)/CC Outputs/Current setpoint value Ch.16 <-> Data Pointer/CurrentSetpointValues[15]
//     Term 45 (AT2202-0500)/CC Outputs/Current setpoint value Ch.17 <-> Data Pointer/CurrentSetpointValues[16]
//     Term 45 (AT2202-0500)/CC Outputs/Current setpoint value Ch.18 <-> Data Pointer/CurrentSetpointValues[17]
//     Term 45 (AT2202-0500)/CC Outputs/Current setpoint value Ch.19 <-> Data Pointer/CurrentSetpointValues[18]
//     Term 45 (AT2202-0500)/CC Outputs/Current setpoint value Ch.2 <-> Data Pointer/CurrentSetpointValues[1]
//     Term 45 (AT2202-0500)/CC Outputs/Current setpoint value Ch.20 <-> Data Pointer/CurrentSetpointValues[19]
//     Term 45 (AT2202-0500)/CC Outputs/Current setpoint value Ch.21 <-> Data Pointer/CurrentSetpointValues[20]
//     Term 45 (AT2202-0500)/CC Outputs/Current setpoint value Ch.22 <-> Data Pointer/CurrentSetpointValues[21]
//     Term 45 (AT2202-0500)/CC Outputs/Current setpoint value Ch.23 <-> Data Pointer/CurrentSetpointValues[22]
//     Term 45 (AT2202-0500)/CC Outputs/Current setpoint value Ch.24 <-> Data Pointer/CurrentSetpointValues[23]
//     Term 45 (AT2202-0500)/CC Outputs/Current setpoint value Ch.25 <-> Data Pointer/CurrentSetpointValues[24]
//     Term 45 (AT2202-0500)/CC Outputs/Current setpoint value Ch.26 <-> Data Pointer/CurrentSetpointValues[25]
//     Term 45 (AT2202-0500)/CC Outputs/Current setpoint value Ch.27 <-> Data Pointer/CurrentSetpointValues[26]
//     Term 45 (AT2202-0500)/CC Outputs/Current setpoint value Ch.28 <-> Data Pointer/CurrentSetpointValues[27]
//     Term 45 (AT2202-0500)/CC Outputs/Current setpoint value Ch.29 <-> Data Pointer/CurrentSetpointValues[28]
//     Term 45 (AT2202-0500)/CC Outputs/Current setpoint value Ch.3 <-> Data Pointer/CurrentSetpointValues[2]
//     Term 45 (AT2202-0500)/CC Outputs/Current setpoint value Ch.30 <-> Data Pointer/CurrentSetpointValues[29]
//     Term 45 (AT2202-0500)/CC Outputs/Current setpoint value Ch.4 <-> Data Pointer/CurrentSetpointValues[3]
//     Term 45 (AT2202-0500)/CC Outputs/Current setpoint value Ch.5 <-> Data Pointer/CurrentSetpointValues[4]
//     Term 45 (AT2202-0500)/CC Outputs/Current setpoint value Ch.6 <-> Data Pointer/CurrentSetpointValues[5]
//     Term 45 (AT2202-0500)/CC Outputs/Current setpoint value Ch.7 <-> Data Pointer/CurrentSetpointValues[6]
//     Term 45 (AT2202-0500)/CC Outputs/Current setpoint value Ch.8 <-> Data Pointer/CurrentSetpointValues[7]
//     Term 45 (AT2202-0500)/CC Outputs/Current setpoint value Ch.9 <-> Data Pointer/CurrentSetpointValues[8]
//     Term 45 (AT2202-0500)/LFB Inputs/BinaryData <-> Data Pointer/HallSensorValues
//   Device 27 <-> TcCOM Objects/XTS ProcessingUnit 1/Part 1/Module 36
//     Term 46 (AT2200-0500)/CC Inputs/Current actual value Ch.1 <-> Data Pointer/CurrentActualValues[0]
//     Term 46 (AT2200-0500)/CC Inputs/Current actual value Ch.10 <-> Data Pointer/CurrentActualValues[9]
//     Term 46 (AT2200-0500)/CC Inputs/Current actual value Ch.11 <-> Data Pointer/CurrentActualValues[10]
//     Term 46 (AT2200-0500)/CC Inputs/Current actual value Ch.12 <-> Data Pointer/CurrentActualValues[11]
//     Term 46 (AT2200-0500)/CC Inputs/Current actual value Ch.13 <-> Data Pointer/CurrentActualValues[12]
//     Term 46 (AT2200-0500)/CC Inputs/Current actual value Ch.14 <-> Data Pointer/CurrentActualValues[13]
//     Term 46 (AT2200-0500)/CC Inputs/Current actual value Ch.15 <-> Data Pointer/CurrentActualValues[14]
//     Term 46 (AT2200-0500)/CC Inputs/Current actual value Ch.16 <-> Data Pointer/CurrentActualValues[15]
//     Term 46 (AT2200-0500)/CC Inputs/Current actual value Ch.17 <-> Data Pointer/CurrentActualValues[16]
//     Term 46 (AT2200-0500)/CC Inputs/Current actual value Ch.18 <-> Data Pointer/CurrentActualValues[17]
//     Term 46 (AT2200-0500)/CC Inputs/Current actual value Ch.19 <-> Data Pointer/CurrentActualValues[18]
//     Term 46 (AT2200-0500)/CC Inputs/Current actual value Ch.2 <-> Data Pointer/CurrentActualValues[1]
//     Term 46 (AT2200-0500)/CC Inputs/Current actual value Ch.20 <-> Data Pointer/CurrentActualValues[19]
//     Term 46 (AT2200-0500)/CC Inputs/Current actual value Ch.21 <-> Data Pointer/CurrentActualValues[20]
//     Term 46 (AT2200-0500)/CC Inputs/Current actual value Ch.22 <-> Data Pointer/CurrentActualValues[21]
//     Term 46 (AT2200-0500)/CC Inputs/Current actual value Ch.23 <-> Data Pointer/CurrentActualValues[22]
//     Term 46 (AT2200-0500)/CC Inputs/Current actual value Ch.24 <-> Data Pointer/CurrentActualValues[23]
//     Term 46 (AT2200-0500)/CC Inputs/Current actual value Ch.25 <-> Data Pointer/CurrentActualValues[24]
//     Term 46 (AT2200-0500)/CC Inputs/Current actual value Ch.26 <-> Data Pointer/CurrentActualValues[25]
//     Term 46 (AT2200-0500)/CC Inputs/Current actual value Ch.27 <-> Data Pointer/CurrentActualValues[26]
//     Term 46 (AT2200-0500)/CC Inputs/Current actual value Ch.28 <-> Data Pointer/CurrentActualValues[27]
//     Term 46 (AT2200-0500)/CC Inputs/Current actual value Ch.29 <-> Data Pointer/CurrentActualValues[28]
//     Term 46 (AT2200-0500)/CC Inputs/Current actual value Ch.3 <-> Data Pointer/CurrentActualValues[2]
//     Term 46 (AT2200-0500)/CC Inputs/Current actual value Ch.30 <-> Data Pointer/CurrentActualValues[29]
//     Term 46 (AT2200-0500)/CC Inputs/Current actual value Ch.4 <-> Data Pointer/CurrentActualValues[3]
//     Term 46 (AT2200-0500)/CC Inputs/Current actual value Ch.5 <-> Data Pointer/CurrentActualValues[4]
//     Term 46 (AT2200-0500)/CC Inputs/Current actual value Ch.6 <-> Data Pointer/CurrentActualValues[5]
//     Term 46 (AT2200-0500)/CC Inputs/Current actual value Ch.7 <-> Data Pointer/CurrentActualValues[6]
//     Term 46 (AT2200-0500)/CC Inputs/Current actual value Ch.8 <-> Data Pointer/CurrentActualValues[7]
//     Term 46 (AT2200-0500)/CC Inputs/Current actual value Ch.9 <-> Data Pointer/CurrentActualValues[8]
//     Term 46 (AT2200-0500)/CC Inputs/Status <-> Data Pointer/Status
//     Term 46 (AT2200-0500)/CC Outputs/Control <-> Data Pointer/Control
//     Term 46 (AT2200-0500)/CC Outputs/Current setpoint value Ch.1 <-> Data Pointer/CurrentSetpointValues[0]
//     Term 46 (AT2200-0500)/CC Outputs/Current setpoint value Ch.10 <-> Data Pointer/CurrentSetpointValues[9]
//     Term 46 (AT2200-0500)/CC Outputs/Current setpoint value Ch.11 <-> Data Pointer/CurrentSetpointValues[10]
//     Term 46 (AT2200-0500)/CC Outputs/Current setpoint value Ch.12 <-> Data Pointer/CurrentSetpointValues[11]
//     Term 46 (AT2200-0500)/CC Outputs/Current setpoint value Ch.13 <-> Data Pointer/CurrentSetpointValues[12]
//     Term 46 (AT2200-0500)/CC Outputs/Current setpoint value Ch.14 <-> Data Pointer/CurrentSetpointValues[13]
//     Term 46 (AT2200-0500)/CC Outputs/Current setpoint value Ch.15 <-> Data Pointer/CurrentSetpointValues[14]
//     Term 46 (AT2200-0500)/CC Outputs/Current setpoint value Ch.16 <-> Data Pointer/CurrentSetpointValues[15]
//     Term 46 (AT2200-0500)/CC Outputs/Current setpoint value Ch.17 <-> Data Pointer/CurrentSetpointValues[16]
//     Term 46 (AT2200-0500)/CC Outputs/Current setpoint value Ch.18 <-> Data Pointer/CurrentSetpointValues[17]
//     Term 46 (AT2200-0500)/CC Outputs/Current setpoint value Ch.19 <-> Data Pointer/CurrentSetpointValues[18]
//     Term 46 (AT2200-0500)/CC Outputs/Current setpoint value Ch.2 <-> Data Pointer/CurrentSetpointValues[1]
//     Term 46 (AT2200-0500)/CC Outputs/Current setpoint value Ch.20 <-> Data Pointer/CurrentSetpointValues[19]
//     Term 46 (AT2200-0500)/CC Outputs/Current setpoint value Ch.21 <-> Data Pointer/CurrentSetpointValues[20]
//     Term 46 (AT2200-0500)/CC Outputs/Current setpoint value Ch.22 <-> Data Pointer/CurrentSetpointValues[21]
//     Term 46 (AT2200-0500)/CC Outputs/Current setpoint value Ch.23 <-> Data Pointer/CurrentSetpointValues[22]
//     Term 46 (AT2200-0500)/CC Outputs/Current setpoint value Ch.24 <-> Data Pointer/CurrentSetpointValues[23]
//     Term 46 (AT2200-0500)/CC Outputs/Current setpoint value Ch.25 <-> Data Pointer/CurrentSetpointValues[24]
//     Term 46 (AT2200-0500)/CC Outputs/Current setpoint value Ch.26 <-> Data Pointer/CurrentSetpointValues[25]
//     Term 46 (AT2200-0500)/CC Outputs/Current setpoint value Ch.27 <-> Data Pointer/CurrentSetpointValues[26]
//     Term 46 (AT2200-0500)/CC Outputs/Current setpoint value Ch.28 <-> Data Pointer/CurrentSetpointValues[27]
//     Term 46 (AT2200-0500)/CC Outputs/Current setpoint value Ch.29 <-> Data Pointer/CurrentSetpointValues[28]
//     Term 46 (AT2200-0500)/CC Outputs/Current setpoint value Ch.3 <-> Data Pointer/CurrentSetpointValues[2]
//     Term 46 (AT2200-0500)/CC Outputs/Current setpoint value Ch.30 <-> Data Pointer/CurrentSetpointValues[29]
//     Term 46 (AT2200-0500)/CC Outputs/Current setpoint value Ch.4 <-> Data Pointer/CurrentSetpointValues[3]
//     Term 46 (AT2200-0500)/CC Outputs/Current setpoint value Ch.5 <-> Data Pointer/CurrentSetpointValues[4]
//     Term 46 (AT2200-0500)/CC Outputs/Current setpoint value Ch.6 <-> Data Pointer/CurrentSetpointValues[5]
//     Term 46 (AT2200-0500)/CC Outputs/Current setpoint value Ch.7 <-> Data Pointer/CurrentSetpointValues[6]
//     Term 46 (AT2200-0500)/CC Outputs/Current setpoint value Ch.8 <-> Data Pointer/CurrentSetpointValues[7]
//     Term 46 (AT2200-0500)/CC Outputs/Current setpoint value Ch.9 <-> Data Pointer/CurrentSetpointValues[8]
//     Term 46 (AT2200-0500)/LFB Inputs/BinaryData <-> Data Pointer/HallSensorValues
//   Device 27 <-> TcCOM Objects/XTS ProcessingUnit 1/Part 1/Module 37
//     Term 47 (AT2040-0250)/CC Inputs/Current actual value Ch.1 <-> Data Pointer/CurrentActualValues[0]
//     Term 47 (AT2040-0250)/CC Inputs/Current actual value Ch.10 <-> Data Pointer/CurrentActualValues[9]
//     Term 47 (AT2040-0250)/CC Inputs/Current actual value Ch.11 <-> Data Pointer/CurrentActualValues[10]
//     Term 47 (AT2040-0250)/CC Inputs/Current actual value Ch.12 <-> Data Pointer/CurrentActualValues[11]
//     Term 47 (AT2040-0250)/CC Inputs/Current actual value Ch.13 <-> Data Pointer/CurrentActualValues[12]
//     Term 47 (AT2040-0250)/CC Inputs/Current actual value Ch.14 <-> Data Pointer/CurrentActualValues[13]
//     Term 47 (AT2040-0250)/CC Inputs/Current actual value Ch.15 <-> Data Pointer/CurrentActualValues[14]
//     Term 47 (AT2040-0250)/CC Inputs/Current actual value Ch.2 <-> Data Pointer/CurrentActualValues[1]
//     Term 47 (AT2040-0250)/CC Inputs/Current actual value Ch.3 <-> Data Pointer/CurrentActualValues[2]
//     Term 47 (AT2040-0250)/CC Inputs/Current actual value Ch.4 <-> Data Pointer/CurrentActualValues[3]
//     Term 47 (AT2040-0250)/CC Inputs/Current actual value Ch.5 <-> Data Pointer/CurrentActualValues[4]
//     Term 47 (AT2040-0250)/CC Inputs/Current actual value Ch.6 <-> Data Pointer/CurrentActualValues[5]
//     Term 47 (AT2040-0250)/CC Inputs/Current actual value Ch.7 <-> Data Pointer/CurrentActualValues[6]
//     Term 47 (AT2040-0250)/CC Inputs/Current actual value Ch.8 <-> Data Pointer/CurrentActualValues[7]
//     Term 47 (AT2040-0250)/CC Inputs/Current actual value Ch.9 <-> Data Pointer/CurrentActualValues[8]
//     Term 47 (AT2040-0250)/CC Inputs/Status <-> Data Pointer/Status
//     Term 47 (AT2040-0250)/CC Outputs/Control <-> Data Pointer/Control
//     Term 47 (AT2040-0250)/CC Outputs/Current setpoint value Ch.1 <-> Data Pointer/CurrentSetpointValues[0]
//     Term 47 (AT2040-0250)/CC Outputs/Current setpoint value Ch.10 <-> Data Pointer/CurrentSetpointValues[9]
//     Term 47 (AT2040-0250)/CC Outputs/Current setpoint value Ch.11 <-> Data Pointer/CurrentSetpointValues[10]
//     Term 47 (AT2040-0250)/CC Outputs/Current setpoint value Ch.12 <-> Data Pointer/CurrentSetpointValues[11]
//     Term 47 (AT2040-0250)/CC Outputs/Current setpoint value Ch.13 <-> Data Pointer/CurrentSetpointValues[12]
//     Term 47 (AT2040-0250)/CC Outputs/Current setpoint value Ch.14 <-> Data Pointer/CurrentSetpointValues[13]
//     Term 47 (AT2040-0250)/CC Outputs/Current setpoint value Ch.15 <-> Data Pointer/CurrentSetpointValues[14]
//     Term 47 (AT2040-0250)/CC Outputs/Current setpoint value Ch.2 <-> Data Pointer/CurrentSetpointValues[1]
//     Term 47 (AT2040-0250)/CC Outputs/Current setpoint value Ch.3 <-> Data Pointer/CurrentSetpointValues[2]
//     Term 47 (AT2040-0250)/CC Outputs/Current setpoint value Ch.4 <-> Data Pointer/CurrentSetpointValues[3]
//     Term 47 (AT2040-0250)/CC Outputs/Current setpoint value Ch.5 <-> Data Pointer/CurrentSetpointValues[4]
//     Term 47 (AT2040-0250)/CC Outputs/Current setpoint value Ch.6 <-> Data Pointer/CurrentSetpointValues[5]
//     Term 47 (AT2040-0250)/CC Outputs/Current setpoint value Ch.7 <-> Data Pointer/CurrentSetpointValues[6]
//     Term 47 (AT2040-0250)/CC Outputs/Current setpoint value Ch.8 <-> Data Pointer/CurrentSetpointValues[7]
//     Term 47 (AT2040-0250)/CC Outputs/Current setpoint value Ch.9 <-> Data Pointer/CurrentSetpointValues[8]
//     Term 47 (AT2040-0250)/Term 48 (AT2040-5250)/FB Inputs/Value Channel 01 <-> Data Pointer/RawPositionValues[0]
//     Term 47 (AT2040-0250)/Term 48 (AT2040-5250)/FB Inputs/Value Channel 02 <-> Data Pointer/RawPositionValues[1]
//     Term 47 (AT2040-0250)/Term 48 (AT2040-5250)/FB Inputs/Value Channel 03 <-> Data Pointer/RawPositionValues[2]
//     Term 47 (AT2040-0250)/Term 48 (AT2040-5250)/FB Inputs/Value Channel 04 <-> Data Pointer/RawPositionValues[3]
//     Term 47 (AT2040-0250)/Term 48 (AT2040-5250)/FB Inputs/Value Channel 05 <-> Data Pointer/RawPositionValues[4]
//     Term 47 (AT2040-0250)/Term 48 (AT2040-5250)/FB Inputs/Value Channel 06 <-> Data Pointer/RawPositionValues[5]
//     Term 47 (AT2040-0250)/Term 48 (AT2040-5250)/FB Inputs/Value Channel 07 <-> Data Pointer/RawPositionValues[6]
//     Term 47 (AT2040-0250)/Term 48 (AT2040-5250)/FB Inputs/Value Channel 08 <-> Data Pointer/RawPositionValues[7]
//     Term 47 (AT2040-0250)/Term 48 (AT2040-5250)/FB Inputs/Value Channel 09 <-> Data Pointer/RawPositionValues[8]
//     Term 47 (AT2040-0250)/Term 48 (AT2040-5250)/FB Inputs/Value Channel 10 <-> Data Pointer/RawPositionValues[9]
//     Term 47 (AT2040-0250)/Term 48 (AT2040-5250)/FB Inputs/Value Channel 11 <-> Data Pointer/RawPositionValues[10]
//     Term 47 (AT2040-0250)/Term 48 (AT2040-5250)/FB Inputs/Value Channel 12 <-> Data Pointer/RawPositionValues[11]
//     Term 47 (AT2040-0250)/Term 48 (AT2040-5250)/FB Inputs/Value Channel 13 <-> Data Pointer/RawPositionValues[12]
//     Term 47 (AT2040-0250)/Term 48 (AT2040-5250)/FB Inputs/Value Channel 14 <-> Data Pointer/RawPositionValues[13]
//     Term 47 (AT2040-0250)/Term 48 (AT2040-5250)/FB Inputs/Value Channel 15 <-> Data Pointer/RawPositionValues[14]
//     Term 47 (AT2040-0250)/Term 48 (AT2040-5250)/FB Inputs/Value Channel 16 <-> Data Pointer/RawPositionValues[15]
//     Term 47 (AT2040-0250)/Term 48 (AT2040-5250)/FB Inputs/Value Channel 17 <-> Data Pointer/RawPositionValues[16]
//     Term 47 (AT2040-0250)/Term 48 (AT2040-5250)/FB Inputs/Value Channel 18 <-> Data Pointer/RawPositionValues[17]
//     Term 47 (AT2040-0250)/Term 48 (AT2040-5250)/FB Inputs/Value Channel 19 <-> Data Pointer/RawPositionValues[18]
//     Term 47 (AT2040-0250)/Term 48 (AT2040-5250)/FB Inputs/Value Channel 20 <-> Data Pointer/RawPositionValues[19]
//     Term 47 (AT2040-0250)/Term 48 (AT2040-5250)/FB Inputs/Value Channel 21 <-> Data Pointer/RawPositionValues[20]
//     Term 47 (AT2040-0250)/Term 48 (AT2040-5250)/FB Inputs/Value Channel 22 <-> Data Pointer/RawPositionValues[21]
//     Term 47 (AT2040-0250)/Term 48 (AT2040-5250)/FB Inputs/Value Channel 23 <-> Data Pointer/RawPositionValues[22]
//     Term 47 (AT2040-0250)/Term 48 (AT2040-5250)/FB Inputs/Value Channel 24 <-> Data Pointer/RawPositionValues[23]
//     Term 47 (AT2040-0250)/Term 48 (AT2040-5250)/FB Inputs/Value Channel 25 <-> Data Pointer/RawPositionValues[24]
//     Term 47 (AT2040-0250)/Term 48 (AT2040-5250)/FB Inputs/Value Channel 26 <-> Data Pointer/RawPositionValues[25]
//     Term 47 (AT2040-0250)/Term 48 (AT2040-5250)/FB Inputs/Value Channel 27 <-> Data Pointer/RawPositionValues[26]
//     Term 47 (AT2040-0250)/Term 48 (AT2040-5250)/FB Inputs/Value Channel 28 <-> Data Pointer/RawPositionValues[27]
//     Term 47 (AT2040-0250)/Term 48 (AT2040-5250)/FB Inputs/Value Channel 29 <-> Data Pointer/RawPositionValues[28]
//     Term 47 (AT2040-0250)/Term 48 (AT2040-5250)/FB Inputs/Value Channel 30 <-> Data Pointer/RawPositionValues[29]
//     Term 47 (AT2040-0250)/Term 48 (AT2040-5250)/FB Inputs/Value Channel 31 <-> Data Pointer/RawPositionValues[30]
//     Term 47 (AT2040-0250)/Term 48 (AT2040-5250)/FB Inputs/Value Channel 32 <-> Data Pointer/RawPositionValues[31]
//   Device 28 <-> TcCOM Objects/XTS ProcessingUnit 1/Part 1/Module 38
//     Term 49 (AT2042-0250)/CC Inputs/Current actual value Ch.1 <-> Data Pointer/CurrentActualValues[0]
//     Term 49 (AT2042-0250)/CC Inputs/Current actual value Ch.10 <-> Data Pointer/CurrentActualValues[9]
//     Term 49 (AT2042-0250)/CC Inputs/Current actual value Ch.11 <-> Data Pointer/CurrentActualValues[10]
//     Term 49 (AT2042-0250)/CC Inputs/Current actual value Ch.12 <-> Data Pointer/CurrentActualValues[11]
//     Term 49 (AT2042-0250)/CC Inputs/Current actual value Ch.13 <-> Data Pointer/CurrentActualValues[12]
//     Term 49 (AT2042-0250)/CC Inputs/Current actual value Ch.14 <-> Data Pointer/CurrentActualValues[13]
//     Term 49 (AT2042-0250)/CC Inputs/Current actual value Ch.15 <-> Data Pointer/CurrentActualValues[14]
//     Term 49 (AT2042-0250)/CC Inputs/Current actual value Ch.2 <-> Data Pointer/CurrentActualValues[1]
//     Term 49 (AT2042-0250)/CC Inputs/Current actual value Ch.3 <-> Data Pointer/CurrentActualValues[2]
//     Term 49 (AT2042-0250)/CC Inputs/Current actual value Ch.4 <-> Data Pointer/CurrentActualValues[3]
//     Term 49 (AT2042-0250)/CC Inputs/Current actual value Ch.5 <-> Data Pointer/CurrentActualValues[4]
//     Term 49 (AT2042-0250)/CC Inputs/Current actual value Ch.6 <-> Data Pointer/CurrentActualValues[5]
//     Term 49 (AT2042-0250)/CC Inputs/Current actual value Ch.7 <-> Data Pointer/CurrentActualValues[6]
//     Term 49 (AT2042-0250)/CC Inputs/Current actual value Ch.8 <-> Data Pointer/CurrentActualValues[7]
//     Term 49 (AT2042-0250)/CC Inputs/Current actual value Ch.9 <-> Data Pointer/CurrentActualValues[8]
//     Term 49 (AT2042-0250)/CC Inputs/Status <-> Data Pointer/Status
//     Term 49 (AT2042-0250)/CC Outputs/Control <-> Data Pointer/Control
//     Term 49 (AT2042-0250)/CC Outputs/Current setpoint value Ch.1 <-> Data Pointer/CurrentSetpointValues[0]
//     Term 49 (AT2042-0250)/CC Outputs/Current setpoint value Ch.10 <-> Data Pointer/CurrentSetpointValues[9]
//     Term 49 (AT2042-0250)/CC Outputs/Current setpoint value Ch.11 <-> Data Pointer/CurrentSetpointValues[10]
//     Term 49 (AT2042-0250)/CC Outputs/Current setpoint value Ch.12 <-> Data Pointer/CurrentSetpointValues[11]
//     Term 49 (AT2042-0250)/CC Outputs/Current setpoint value Ch.13 <-> Data Pointer/CurrentSetpointValues[12]
//     Term 49 (AT2042-0250)/CC Outputs/Current setpoint value Ch.14 <-> Data Pointer/CurrentSetpointValues[13]
//     Term 49 (AT2042-0250)/CC Outputs/Current setpoint value Ch.15 <-> Data Pointer/CurrentSetpointValues[14]
//     Term 49 (AT2042-0250)/CC Outputs/Current setpoint value Ch.2 <-> Data Pointer/CurrentSetpointValues[1]
//     Term 49 (AT2042-0250)/CC Outputs/Current setpoint value Ch.3 <-> Data Pointer/CurrentSetpointValues[2]
//     Term 49 (AT2042-0250)/CC Outputs/Current setpoint value Ch.4 <-> Data Pointer/CurrentSetpointValues[3]
//     Term 49 (AT2042-0250)/CC Outputs/Current setpoint value Ch.5 <-> Data Pointer/CurrentSetpointValues[4]
//     Term 49 (AT2042-0250)/CC Outputs/Current setpoint value Ch.6 <-> Data Pointer/CurrentSetpointValues[5]
//     Term 49 (AT2042-0250)/CC Outputs/Current setpoint value Ch.7 <-> Data Pointer/CurrentSetpointValues[6]
//     Term 49 (AT2042-0250)/CC Outputs/Current setpoint value Ch.8 <-> Data Pointer/CurrentSetpointValues[7]
//     Term 49 (AT2042-0250)/CC Outputs/Current setpoint value Ch.9 <-> Data Pointer/CurrentSetpointValues[8]
//     Term 49 (AT2042-0250)/Term 50 (AT2042-5250)/FB Inputs/Value Channel 01 <-> Data Pointer/RawPositionValues[0]
//     Term 49 (AT2042-0250)/Term 50 (AT2042-5250)/FB Inputs/Value Channel 02 <-> Data Pointer/RawPositionValues[1]
//     Term 49 (AT2042-0250)/Term 50 (AT2042-5250)/FB Inputs/Value Channel 03 <-> Data Pointer/RawPositionValues[2]
//     Term 49 (AT2042-0250)/Term 50 (AT2042-5250)/FB Inputs/Value Channel 04 <-> Data Pointer/RawPositionValues[3]
//     Term 49 (AT2042-0250)/Term 50 (AT2042-5250)/FB Inputs/Value Channel 05 <-> Data Pointer/RawPositionValues[4]
//     Term 49 (AT2042-0250)/Term 50 (AT2042-5250)/FB Inputs/Value Channel 06 <-> Data Pointer/RawPositionValues[5]
//     Term 49 (AT2042-0250)/Term 50 (AT2042-5250)/FB Inputs/Value Channel 07 <-> Data Pointer/RawPositionValues[6]
//     Term 49 (AT2042-0250)/Term 50 (AT2042-5250)/FB Inputs/Value Channel 08 <-> Data Pointer/RawPositionValues[7]
//     Term 49 (AT2042-0250)/Term 50 (AT2042-5250)/FB Inputs/Value Channel 09 <-> Data Pointer/RawPositionValues[8]
//     Term 49 (AT2042-0250)/Term 50 (AT2042-5250)/FB Inputs/Value Channel 10 <-> Data Pointer/RawPositionValues[9]
//     Term 49 (AT2042-0250)/Term 50 (AT2042-5250)/FB Inputs/Value Channel 11 <-> Data Pointer/RawPositionValues[10]
//     Term 49 (AT2042-0250)/Term 50 (AT2042-5250)/FB Inputs/Value Channel 12 <-> Data Pointer/RawPositionValues[11]
//     Term 49 (AT2042-0250)/Term 50 (AT2042-5250)/FB Inputs/Value Channel 13 <-> Data Pointer/RawPositionValues[12]
//     Term 49 (AT2042-0250)/Term 50 (AT2042-5250)/FB Inputs/Value Channel 14 <-> Data Pointer/RawPositionValues[13]
//     Term 49 (AT2042-0250)/Term 50 (AT2042-5250)/FB Inputs/Value Channel 15 <-> Data Pointer/RawPositionValues[14]
//     Term 49 (AT2042-0250)/Term 50 (AT2042-5250)/FB Inputs/Value Channel 16 <-> Data Pointer/RawPositionValues[15]
//     Term 49 (AT2042-0250)/Term 50 (AT2042-5250)/FB Inputs/Value Channel 17 <-> Data Pointer/RawPositionValues[16]
//     Term 49 (AT2042-0250)/Term 50 (AT2042-5250)/FB Inputs/Value Channel 18 <-> Data Pointer/RawPositionValues[17]
//     Term 49 (AT2042-0250)/Term 50 (AT2042-5250)/FB Inputs/Value Channel 19 <-> Data Pointer/RawPositionValues[18]
//     Term 49 (AT2042-0250)/Term 50 (AT2042-5250)/FB Inputs/Value Channel 20 <-> Data Pointer/RawPositionValues[19]
//     Term 49 (AT2042-0250)/Term 50 (AT2042-5250)/FB Inputs/Value Channel 21 <-> Data Pointer/RawPositionValues[20]
//     Term 49 (AT2042-0250)/Term 50 (AT2042-5250)/FB Inputs/Value Channel 22 <-> Data Pointer/RawPositionValues[21]
//     Term 49 (AT2042-0250)/Term 50 (AT2042-5250)/FB Inputs/Value Channel 23 <-> Data Pointer/RawPositionValues[22]
//     Term 49 (AT2042-0250)/Term 50 (AT2042-5250)/FB Inputs/Value Channel 24 <-> Data Pointer/RawPositionValues[23]
//     Term 49 (AT2042-0250)/Term 50 (AT2042-5250)/FB Inputs/Value Channel 25 <-> Data Pointer/RawPositionValues[24]
//     Term 49 (AT2042-0250)/Term 50 (AT2042-5250)/FB Inputs/Value Channel 26 <-> Data Pointer/RawPositionValues[25]
//     Term 49 (AT2042-0250)/Term 50 (AT2042-5250)/FB Inputs/Value Channel 27 <-> Data Pointer/RawPositionValues[26]
//     Term 49 (AT2042-0250)/Term 50 (AT2042-5250)/FB Inputs/Value Channel 28 <-> Data Pointer/RawPositionValues[27]
//     Term 49 (AT2042-0250)/Term 50 (AT2042-5250)/FB Inputs/Value Channel 29 <-> Data Pointer/RawPositionValues[28]
//     Term 49 (AT2042-0250)/Term 50 (AT2042-5250)/FB Inputs/Value Channel 30 <-> Data Pointer/RawPositionValues[29]
//     Term 49 (AT2042-0250)/Term 50 (AT2042-5250)/FB Inputs/Value Channel 31 <-> Data Pointer/RawPositionValues[30]
//     Term 49 (AT2042-0250)/Term 50 (AT2042-5250)/FB Inputs/Value Channel 32 <-> Data Pointer/RawPositionValues[31]
//   Device 28 <-> TcCOM Objects/XTS ProcessingUnit 1/Part 1/Module 39
//     Term 51 (AT2200-0500)/CC Inputs/Current actual value Ch.1 <-> Data Pointer/CurrentActualValues[0]
//     Term 51 (AT2200-0500)/CC Inputs/Current actual value Ch.10 <-> Data Pointer/CurrentActualValues[9]
//     Term 51 (AT2200-0500)/CC Inputs/Current actual value Ch.11 <-> Data Pointer/CurrentActualValues[10]
//     Term 51 (AT2200-0500)/CC Inputs/Current actual value Ch.12 <-> Data Pointer/CurrentActualValues[11]
//     Term 51 (AT2200-0500)/CC Inputs/Current actual value Ch.13 <-> Data Pointer/CurrentActualValues[12]
//     Term 51 (AT2200-0500)/CC Inputs/Current actual value Ch.14 <-> Data Pointer/CurrentActualValues[13]
//     Term 51 (AT2200-0500)/CC Inputs/Current actual value Ch.15 <-> Data Pointer/CurrentActualValues[14]
//     Term 51 (AT2200-0500)/CC Inputs/Current actual value Ch.16 <-> Data Pointer/CurrentActualValues[15]
//     Term 51 (AT2200-0500)/CC Inputs/Current actual value Ch.17 <-> Data Pointer/CurrentActualValues[16]
//     Term 51 (AT2200-0500)/CC Inputs/Current actual value Ch.18 <-> Data Pointer/CurrentActualValues[17]
//     Term 51 (AT2200-0500)/CC Inputs/Current actual value Ch.19 <-> Data Pointer/CurrentActualValues[18]
//     Term 51 (AT2200-0500)/CC Inputs/Current actual value Ch.2 <-> Data Pointer/CurrentActualValues[1]
//     Term 51 (AT2200-0500)/CC Inputs/Current actual value Ch.20 <-> Data Pointer/CurrentActualValues[19]
//     Term 51 (AT2200-0500)/CC Inputs/Current actual value Ch.21 <-> Data Pointer/CurrentActualValues[20]
//     Term 51 (AT2200-0500)/CC Inputs/Current actual value Ch.22 <-> Data Pointer/CurrentActualValues[21]
//     Term 51 (AT2200-0500)/CC Inputs/Current actual value Ch.23 <-> Data Pointer/CurrentActualValues[22]
//     Term 51 (AT2200-0500)/CC Inputs/Current actual value Ch.24 <-> Data Pointer/CurrentActualValues[23]
//     Term 51 (AT2200-0500)/CC Inputs/Current actual value Ch.25 <-> Data Pointer/CurrentActualValues[24]
//     Term 51 (AT2200-0500)/CC Inputs/Current actual value Ch.26 <-> Data Pointer/CurrentActualValues[25]
//     Term 51 (AT2200-0500)/CC Inputs/Current actual value Ch.27 <-> Data Pointer/CurrentActualValues[26]
//     Term 51 (AT2200-0500)/CC Inputs/Current actual value Ch.28 <-> Data Pointer/CurrentActualValues[27]
//     Term 51 (AT2200-0500)/CC Inputs/Current actual value Ch.29 <-> Data Pointer/CurrentActualValues[28]
//     Term 51 (AT2200-0500)/CC Inputs/Current actual value Ch.3 <-> Data Pointer/CurrentActualValues[2]
//     Term 51 (AT2200-0500)/CC Inputs/Current actual value Ch.30 <-> Data Pointer/CurrentActualValues[29]
//     Term 51 (AT2200-0500)/CC Inputs/Current actual value Ch.4 <-> Data Pointer/CurrentActualValues[3]
//     Term 51 (AT2200-0500)/CC Inputs/Current actual value Ch.5 <-> Data Pointer/CurrentActualValues[4]
//     Term 51 (AT2200-0500)/CC Inputs/Current actual value Ch.6 <-> Data Pointer/CurrentActualValues[5]
//     Term 51 (AT2200-0500)/CC Inputs/Current actual value Ch.7 <-> Data Pointer/CurrentActualValues[6]
//     Term 51 (AT2200-0500)/CC Inputs/Current actual value Ch.8 <-> Data Pointer/CurrentActualValues[7]
//     Term 51 (AT2200-0500)/CC Inputs/Current actual value Ch.9 <-> Data Pointer/CurrentActualValues[8]
//     Term 51 (AT2200-0500)/CC Inputs/Status <-> Data Pointer/Status
//     Term 51 (AT2200-0500)/CC Outputs/Control <-> Data Pointer/Control
//     Term 51 (AT2200-0500)/CC Outputs/Current setpoint value Ch.1 <-> Data Pointer/CurrentSetpointValues[0]
//     Term 51 (AT2200-0500)/CC Outputs/Current setpoint value Ch.10 <-> Data Pointer/CurrentSetpointValues[9]
//     Term 51 (AT2200-0500)/CC Outputs/Current setpoint value Ch.11 <-> Data Pointer/CurrentSetpointValues[10]
//     Term 51 (AT2200-0500)/CC Outputs/Current setpoint value Ch.12 <-> Data Pointer/CurrentSetpointValues[11]
//     Term 51 (AT2200-0500)/CC Outputs/Current setpoint value Ch.13 <-> Data Pointer/CurrentSetpointValues[12]
//     Term 51 (AT2200-0500)/CC Outputs/Current setpoint value Ch.14 <-> Data Pointer/CurrentSetpointValues[13]
//     Term 51 (AT2200-0500)/CC Outputs/Current setpoint value Ch.15 <-> Data Pointer/CurrentSetpointValues[14]
//     Term 51 (AT2200-0500)/CC Outputs/Current setpoint value Ch.16 <-> Data Pointer/CurrentSetpointValues[15]
//     Term 51 (AT2200-0500)/CC Outputs/Current setpoint value Ch.17 <-> Data Pointer/CurrentSetpointValues[16]
//     Term 51 (AT2200-0500)/CC Outputs/Current setpoint value Ch.18 <-> Data Pointer/CurrentSetpointValues[17]
//     Term 51 (AT2200-0500)/CC Outputs/Current setpoint value Ch.19 <-> Data Pointer/CurrentSetpointValues[18]
//     Term 51 (AT2200-0500)/CC Outputs/Current setpoint value Ch.2 <-> Data Pointer/CurrentSetpointValues[1]
//     Term 51 (AT2200-0500)/CC Outputs/Current setpoint value Ch.20 <-> Data Pointer/CurrentSetpointValues[19]
//     Term 51 (AT2200-0500)/CC Outputs/Current setpoint value Ch.21 <-> Data Pointer/CurrentSetpointValues[20]
//     Term 51 (AT2200-0500)/CC Outputs/Current setpoint value Ch.22 <-> Data Pointer/CurrentSetpointValues[21]
//     Term 51 (AT2200-0500)/CC Outputs/Current setpoint value Ch.23 <-> Data Pointer/CurrentSetpointValues[22]
//     Term 51 (AT2200-0500)/CC Outputs/Current setpoint value Ch.24 <-> Data Pointer/CurrentSetpointValues[23]
//     Term 51 (AT2200-0500)/CC Outputs/Current setpoint value Ch.25 <-> Data Pointer/CurrentSetpointValues[24]
//     Term 51 (AT2200-0500)/CC Outputs/Current setpoint value Ch.26 <-> Data Pointer/CurrentSetpointValues[25]
//     Term 51 (AT2200-0500)/CC Outputs/Current setpoint value Ch.27 <-> Data Pointer/CurrentSetpointValues[26]
//     Term 51 (AT2200-0500)/CC Outputs/Current setpoint value Ch.28 <-> Data Pointer/CurrentSetpointValues[27]
//     Term 51 (AT2200-0500)/CC Outputs/Current setpoint value Ch.29 <-> Data Pointer/CurrentSetpointValues[28]
//     Term 51 (AT2200-0500)/CC Outputs/Current setpoint value Ch.3 <-> Data Pointer/CurrentSetpointValues[2]
//     Term 51 (AT2200-0500)/CC Outputs/Current setpoint value Ch.30 <-> Data Pointer/CurrentSetpointValues[29]
//     Term 51 (AT2200-0500)/CC Outputs/Current setpoint value Ch.4 <-> Data Pointer/CurrentSetpointValues[3]
//     Term 51 (AT2200-0500)/CC Outputs/Current setpoint value Ch.5 <-> Data Pointer/CurrentSetpointValues[4]
//     Term 51 (AT2200-0500)/CC Outputs/Current setpoint value Ch.6 <-> Data Pointer/CurrentSetpointValues[5]
//     Term 51 (AT2200-0500)/CC Outputs/Current setpoint value Ch.7 <-> Data Pointer/CurrentSetpointValues[6]
//     Term 51 (AT2200-0500)/CC Outputs/Current setpoint value Ch.8 <-> Data Pointer/CurrentSetpointValues[7]
//     Term 51 (AT2200-0500)/CC Outputs/Current setpoint value Ch.9 <-> Data Pointer/CurrentSetpointValues[8]
//     Term 51 (AT2200-0500)/LFB Inputs/BinaryData <-> Data Pointer/HallSensorValues
//   Device 28 <-> TcCOM Objects/XTS ProcessingUnit 1/Part 1/Module 40
//     Term 52 (AT2200-0500)/CC Inputs/Current actual value Ch.1 <-> Data Pointer/CurrentActualValues[0]
//     Term 52 (AT2200-0500)/CC Inputs/Current actual value Ch.10 <-> Data Pointer/CurrentActualValues[9]
//     Term 52 (AT2200-0500)/CC Inputs/Current actual value Ch.11 <-> Data Pointer/CurrentActualValues[10]
//     Term 52 (AT2200-0500)/CC Inputs/Current actual value Ch.12 <-> Data Pointer/CurrentActualValues[11]
//     Term 52 (AT2200-0500)/CC Inputs/Current actual value Ch.13 <-> Data Pointer/CurrentActualValues[12]
//     Term 52 (AT2200-0500)/CC Inputs/Current actual value Ch.14 <-> Data Pointer/CurrentActualValues[13]
//     Term 52 (AT2200-0500)/CC Inputs/Current actual value Ch.15 <-> Data Pointer/CurrentActualValues[14]
//     Term 52 (AT2200-0500)/CC Inputs/Current actual value Ch.16 <-> Data Pointer/CurrentActualValues[15]
//     Term 52 (AT2200-0500)/CC Inputs/Current actual value Ch.17 <-> Data Pointer/CurrentActualValues[16]
//     Term 52 (AT2200-0500)/CC Inputs/Current actual value Ch.18 <-> Data Pointer/CurrentActualValues[17]
//     Term 52 (AT2200-0500)/CC Inputs/Current actual value Ch.19 <-> Data Pointer/CurrentActualValues[18]
//     Term 52 (AT2200-0500)/CC Inputs/Current actual value Ch.2 <-> Data Pointer/CurrentActualValues[1]
//     Term 52 (AT2200-0500)/CC Inputs/Current actual value Ch.20 <-> Data Pointer/CurrentActualValues[19]
//     Term 52 (AT2200-0500)/CC Inputs/Current actual value Ch.21 <-> Data Pointer/CurrentActualValues[20]
//     Term 52 (AT2200-0500)/CC Inputs/Current actual value Ch.22 <-> Data Pointer/CurrentActualValues[21]
//     Term 52 (AT2200-0500)/CC Inputs/Current actual value Ch.23 <-> Data Pointer/CurrentActualValues[22]
//     Term 52 (AT2200-0500)/CC Inputs/Current actual value Ch.24 <-> Data Pointer/CurrentActualValues[23]
//     Term 52 (AT2200-0500)/CC Inputs/Current actual value Ch.25 <-> Data Pointer/CurrentActualValues[24]
//     Term 52 (AT2200-0500)/CC Inputs/Current actual value Ch.26 <-> Data Pointer/CurrentActualValues[25]
//     Term 52 (AT2200-0500)/CC Inputs/Current actual value Ch.27 <-> Data Pointer/CurrentActualValues[26]
//     Term 52 (AT2200-0500)/CC Inputs/Current actual value Ch.28 <-> Data Pointer/CurrentActualValues[27]
//     Term 52 (AT2200-0500)/CC Inputs/Current actual value Ch.29 <-> Data Pointer/CurrentActualValues[28]
//     Term 52 (AT2200-0500)/CC Inputs/Current actual value Ch.3 <-> Data Pointer/CurrentActualValues[2]
//     Term 52 (AT2200-0500)/CC Inputs/Current actual value Ch.30 <-> Data Pointer/CurrentActualValues[29]
//     Term 52 (AT2200-0500)/CC Inputs/Current actual value Ch.4 <-> Data Pointer/CurrentActualValues[3]
//     Term 52 (AT2200-0500)/CC Inputs/Current actual value Ch.5 <-> Data Pointer/CurrentActualValues[4]
//     Term 52 (AT2200-0500)/CC Inputs/Current actual value Ch.6 <-> Data Pointer/CurrentActualValues[5]
//     Term 52 (AT2200-0500)/CC Inputs/Current actual value Ch.7 <-> Data Pointer/CurrentActualValues[6]
//     Term 52 (AT2200-0500)/CC Inputs/Current actual value Ch.8 <-> Data Pointer/CurrentActualValues[7]
//     Term 52 (AT2200-0500)/CC Inputs/Current actual value Ch.9 <-> Data Pointer/CurrentActualValues[8]
//     Term 52 (AT2200-0500)/CC Inputs/Status <-> Data Pointer/Status
//     Term 52 (AT2200-0500)/CC Outputs/Control <-> Data Pointer/Control
//     Term 52 (AT2200-0500)/CC Outputs/Current setpoint value Ch.1 <-> Data Pointer/CurrentSetpointValues[0]
//     Term 52 (AT2200-0500)/CC Outputs/Current setpoint value Ch.10 <-> Data Pointer/CurrentSetpointValues[9]
//     Term 52 (AT2200-0500)/CC Outputs/Current setpoint value Ch.11 <-> Data Pointer/CurrentSetpointValues[10]
//     Term 52 (AT2200-0500)/CC Outputs/Current setpoint value Ch.12 <-> Data Pointer/CurrentSetpointValues[11]
//     Term 52 (AT2200-0500)/CC Outputs/Current setpoint value Ch.13 <-> Data Pointer/CurrentSetpointValues[12]
//     Term 52 (AT2200-0500)/CC Outputs/Current setpoint value Ch.14 <-> Data Pointer/CurrentSetpointValues[13]
//     Term 52 (AT2200-0500)/CC Outputs/Current setpoint value Ch.15 <-> Data Pointer/CurrentSetpointValues[14]
//     Term 52 (AT2200-0500)/CC Outputs/Current setpoint value Ch.16 <-> Data Pointer/CurrentSetpointValues[15]
//     Term 52 (AT2200-0500)/CC Outputs/Current setpoint value Ch.17 <-> Data Pointer/CurrentSetpointValues[16]
//     Term 52 (AT2200-0500)/CC Outputs/Current setpoint value Ch.18 <-> Data Pointer/CurrentSetpointValues[17]
//     Term 52 (AT2200-0500)/CC Outputs/Current setpoint value Ch.19 <-> Data Pointer/CurrentSetpointValues[18]
//     Term 52 (AT2200-0500)/CC Outputs/Current setpoint value Ch.2 <-> Data Pointer/CurrentSetpointValues[1]
//     Term 52 (AT2200-0500)/CC Outputs/Current setpoint value Ch.20 <-> Data Pointer/CurrentSetpointValues[19]
//     Term 52 (AT2200-0500)/CC Outputs/Current setpoint value Ch.21 <-> Data Pointer/CurrentSetpointValues[20]
//     Term 52 (AT2200-0500)/CC Outputs/Current setpoint value Ch.22 <-> Data Pointer/CurrentSetpointValues[21]
//     Term 52 (AT2200-0500)/CC Outputs/Current setpoint value Ch.23 <-> Data Pointer/CurrentSetpointValues[22]
//     Term 52 (AT2200-0500)/CC Outputs/Current setpoint value Ch.24 <-> Data Pointer/CurrentSetpointValues[23]
//     Term 52 (AT2200-0500)/CC Outputs/Current setpoint value Ch.25 <-> Data Pointer/CurrentSetpointValues[24]
//     Term 52 (AT2200-0500)/CC Outputs/Current setpoint value Ch.26 <-> Data Pointer/CurrentSetpointValues[25]
//     Term 52 (AT2200-0500)/CC Outputs/Current setpoint value Ch.27 <-> Data Pointer/CurrentSetpointValues[26]
//     Term 52 (AT2200-0500)/CC Outputs/Current setpoint value Ch.28 <-> Data Pointer/CurrentSetpointValues[27]
//     Term 52 (AT2200-0500)/CC Outputs/Current setpoint value Ch.29 <-> Data Pointer/CurrentSetpointValues[28]
//     Term 52 (AT2200-0500)/CC Outputs/Current setpoint value Ch.3 <-> Data Pointer/CurrentSetpointValues[2]
//     Term 52 (AT2200-0500)/CC Outputs/Current setpoint value Ch.30 <-> Data Pointer/CurrentSetpointValues[29]
//     Term 52 (AT2200-0500)/CC Outputs/Current setpoint value Ch.4 <-> Data Pointer/CurrentSetpointValues[3]
//     Term 52 (AT2200-0500)/CC Outputs/Current setpoint value Ch.5 <-> Data Pointer/CurrentSetpointValues[4]
//     Term 52 (AT2200-0500)/CC Outputs/Current setpoint value Ch.6 <-> Data Pointer/CurrentSetpointValues[5]
//     Term 52 (AT2200-0500)/CC Outputs/Current setpoint value Ch.7 <-> Data Pointer/CurrentSetpointValues[6]
//     Term 52 (AT2200-0500)/CC Outputs/Current setpoint value Ch.8 <-> Data Pointer/CurrentSetpointValues[7]
//     Term 52 (AT2200-0500)/CC Outputs/Current setpoint value Ch.9 <-> Data Pointer/CurrentSetpointValues[8]
//     Term 52 (AT2200-0500)/LFB Inputs/BinaryData <-> Data Pointer/HallSensorValues
//   Device 29 <-> TcCOM Objects/XTS ProcessingUnit 1/Part 1/Module 41
//     Term 53 (AT2202-0500)/CC Inputs/Current actual value Ch.1 <-> Data Pointer/CurrentActualValues[0]
//     Term 53 (AT2202-0500)/CC Inputs/Current actual value Ch.10 <-> Data Pointer/CurrentActualValues[9]
//     Term 53 (AT2202-0500)/CC Inputs/Current actual value Ch.11 <-> Data Pointer/CurrentActualValues[10]
//     Term 53 (AT2202-0500)/CC Inputs/Current actual value Ch.12 <-> Data Pointer/CurrentActualValues[11]
//     Term 53 (AT2202-0500)/CC Inputs/Current actual value Ch.13 <-> Data Pointer/CurrentActualValues[12]
//     Term 53 (AT2202-0500)/CC Inputs/Current actual value Ch.14 <-> Data Pointer/CurrentActualValues[13]
//     Term 53 (AT2202-0500)/CC Inputs/Current actual value Ch.15 <-> Data Pointer/CurrentActualValues[14]
//     Term 53 (AT2202-0500)/CC Inputs/Current actual value Ch.16 <-> Data Pointer/CurrentActualValues[15]
//     Term 53 (AT2202-0500)/CC Inputs/Current actual value Ch.17 <-> Data Pointer/CurrentActualValues[16]
//     Term 53 (AT2202-0500)/CC Inputs/Current actual value Ch.18 <-> Data Pointer/CurrentActualValues[17]
//     Term 53 (AT2202-0500)/CC Inputs/Current actual value Ch.19 <-> Data Pointer/CurrentActualValues[18]
//     Term 53 (AT2202-0500)/CC Inputs/Current actual value Ch.2 <-> Data Pointer/CurrentActualValues[1]
//     Term 53 (AT2202-0500)/CC Inputs/Current actual value Ch.20 <-> Data Pointer/CurrentActualValues[19]
//     Term 53 (AT2202-0500)/CC Inputs/Current actual value Ch.21 <-> Data Pointer/CurrentActualValues[20]
//     Term 53 (AT2202-0500)/CC Inputs/Current actual value Ch.22 <-> Data Pointer/CurrentActualValues[21]
//     Term 53 (AT2202-0500)/CC Inputs/Current actual value Ch.23 <-> Data Pointer/CurrentActualValues[22]
//     Term 53 (AT2202-0500)/CC Inputs/Current actual value Ch.24 <-> Data Pointer/CurrentActualValues[23]
//     Term 53 (AT2202-0500)/CC Inputs/Current actual value Ch.25 <-> Data Pointer/CurrentActualValues[24]
//     Term 53 (AT2202-0500)/CC Inputs/Current actual value Ch.26 <-> Data Pointer/CurrentActualValues[25]
//     Term 53 (AT2202-0500)/CC Inputs/Current actual value Ch.27 <-> Data Pointer/CurrentActualValues[26]
//     Term 53 (AT2202-0500)/CC Inputs/Current actual value Ch.28 <-> Data Pointer/CurrentActualValues[27]
//     Term 53 (AT2202-0500)/CC Inputs/Current actual value Ch.29 <-> Data Pointer/CurrentActualValues[28]
//     Term 53 (AT2202-0500)/CC Inputs/Current actual value Ch.3 <-> Data Pointer/CurrentActualValues[2]
//     Term 53 (AT2202-0500)/CC Inputs/Current actual value Ch.30 <-> Data Pointer/CurrentActualValues[29]
//     Term 53 (AT2202-0500)/CC Inputs/Current actual value Ch.4 <-> Data Pointer/CurrentActualValues[3]
//     Term 53 (AT2202-0500)/CC Inputs/Current actual value Ch.5 <-> Data Pointer/CurrentActualValues[4]
//     Term 53 (AT2202-0500)/CC Inputs/Current actual value Ch.6 <-> Data Pointer/CurrentActualValues[5]
//     Term 53 (AT2202-0500)/CC Inputs/Current actual value Ch.7 <-> Data Pointer/CurrentActualValues[6]
//     Term 53 (AT2202-0500)/CC Inputs/Current actual value Ch.8 <-> Data Pointer/CurrentActualValues[7]
//     Term 53 (AT2202-0500)/CC Inputs/Current actual value Ch.9 <-> Data Pointer/CurrentActualValues[8]
//     Term 53 (AT2202-0500)/CC Inputs/Status <-> Data Pointer/Status
//     Term 53 (AT2202-0500)/CC Outputs/Control <-> Data Pointer/Control
//     Term 53 (AT2202-0500)/CC Outputs/Current setpoint value Ch.1 <-> Data Pointer/CurrentSetpointValues[0]
//     Term 53 (AT2202-0500)/CC Outputs/Current setpoint value Ch.10 <-> Data Pointer/CurrentSetpointValues[9]
//     Term 53 (AT2202-0500)/CC Outputs/Current setpoint value Ch.11 <-> Data Pointer/CurrentSetpointValues[10]
//     Term 53 (AT2202-0500)/CC Outputs/Current setpoint value Ch.12 <-> Data Pointer/CurrentSetpointValues[11]
//     Term 53 (AT2202-0500)/CC Outputs/Current setpoint value Ch.13 <-> Data Pointer/CurrentSetpointValues[12]
//     Term 53 (AT2202-0500)/CC Outputs/Current setpoint value Ch.14 <-> Data Pointer/CurrentSetpointValues[13]
//     Term 53 (AT2202-0500)/CC Outputs/Current setpoint value Ch.15 <-> Data Pointer/CurrentSetpointValues[14]
//     Term 53 (AT2202-0500)/CC Outputs/Current setpoint value Ch.16 <-> Data Pointer/CurrentSetpointValues[15]
//     Term 53 (AT2202-0500)/CC Outputs/Current setpoint value Ch.17 <-> Data Pointer/CurrentSetpointValues[16]
//     Term 53 (AT2202-0500)/CC Outputs/Current setpoint value Ch.18 <-> Data Pointer/CurrentSetpointValues[17]
//     Term 53 (AT2202-0500)/CC Outputs/Current setpoint value Ch.19 <-> Data Pointer/CurrentSetpointValues[18]
//     Term 53 (AT2202-0500)/CC Outputs/Current setpoint value Ch.2 <-> Data Pointer/CurrentSetpointValues[1]
//     Term 53 (AT2202-0500)/CC Outputs/Current setpoint value Ch.20 <-> Data Pointer/CurrentSetpointValues[19]
//     Term 53 (AT2202-0500)/CC Outputs/Current setpoint value Ch.21 <-> Data Pointer/CurrentSetpointValues[20]
//     Term 53 (AT2202-0500)/CC Outputs/Current setpoint value Ch.22 <-> Data Pointer/CurrentSetpointValues[21]
//     Term 53 (AT2202-0500)/CC Outputs/Current setpoint value Ch.23 <-> Data Pointer/CurrentSetpointValues[22]
//     Term 53 (AT2202-0500)/CC Outputs/Current setpoint value Ch.24 <-> Data Pointer/CurrentSetpointValues[23]
//     Term 53 (AT2202-0500)/CC Outputs/Current setpoint value Ch.25 <-> Data Pointer/CurrentSetpointValues[24]
//     Term 53 (AT2202-0500)/CC Outputs/Current setpoint value Ch.26 <-> Data Pointer/CurrentSetpointValues[25]
//     Term 53 (AT2202-0500)/CC Outputs/Current setpoint value Ch.27 <-> Data Pointer/CurrentSetpointValues[26]
//     Term 53 (AT2202-0500)/CC Outputs/Current setpoint value Ch.28 <-> Data Pointer/CurrentSetpointValues[27]
//     Term 53 (AT2202-0500)/CC Outputs/Current setpoint value Ch.29 <-> Data Pointer/CurrentSetpointValues[28]
//     Term 53 (AT2202-0500)/CC Outputs/Current setpoint value Ch.3 <-> Data Pointer/CurrentSetpointValues[2]
//     Term 53 (AT2202-0500)/CC Outputs/Current setpoint value Ch.30 <-> Data Pointer/CurrentSetpointValues[29]
//     Term 53 (AT2202-0500)/CC Outputs/Current setpoint value Ch.4 <-> Data Pointer/CurrentSetpointValues[3]
//     Term 53 (AT2202-0500)/CC Outputs/Current setpoint value Ch.5 <-> Data Pointer/CurrentSetpointValues[4]
//     Term 53 (AT2202-0500)/CC Outputs/Current setpoint value Ch.6 <-> Data Pointer/CurrentSetpointValues[5]
//     Term 53 (AT2202-0500)/CC Outputs/Current setpoint value Ch.7 <-> Data Pointer/CurrentSetpointValues[6]
//     Term 53 (AT2202-0500)/CC Outputs/Current setpoint value Ch.8 <-> Data Pointer/CurrentSetpointValues[7]
//     Term 53 (AT2202-0500)/CC Outputs/Current setpoint value Ch.9 <-> Data Pointer/CurrentSetpointValues[8]
//     Term 53 (AT2202-0500)/LFB Inputs/BinaryData <-> Data Pointer/HallSensorValues
//   Device 29 <-> TcCOM Objects/XTS ProcessingUnit 1/Part 1/Module 42
//     Term 54 (AT2200-0500)/CC Inputs/Current actual value Ch.1 <-> Data Pointer/CurrentActualValues[0]
//     Term 54 (AT2200-0500)/CC Inputs/Current actual value Ch.10 <-> Data Pointer/CurrentActualValues[9]
//     Term 54 (AT2200-0500)/CC Inputs/Current actual value Ch.11 <-> Data Pointer/CurrentActualValues[10]
//     Term 54 (AT2200-0500)/CC Inputs/Current actual value Ch.12 <-> Data Pointer/CurrentActualValues[11]
//     Term 54 (AT2200-0500)/CC Inputs/Current actual value Ch.13 <-> Data Pointer/CurrentActualValues[12]
//     Term 54 (AT2200-0500)/CC Inputs/Current actual value Ch.14 <-> Data Pointer/CurrentActualValues[13]
//     Term 54 (AT2200-0500)/CC Inputs/Current actual value Ch.15 <-> Data Pointer/CurrentActualValues[14]
//     Term 54 (AT2200-0500)/CC Inputs/Current actual value Ch.16 <-> Data Pointer/CurrentActualValues[15]
//     Term 54 (AT2200-0500)/CC Inputs/Current actual value Ch.17 <-> Data Pointer/CurrentActualValues[16]
//     Term 54 (AT2200-0500)/CC Inputs/Current actual value Ch.18 <-> Data Pointer/CurrentActualValues[17]
//     Term 54 (AT2200-0500)/CC Inputs/Current actual value Ch.19 <-> Data Pointer/CurrentActualValues[18]
//     Term 54 (AT2200-0500)/CC Inputs/Current actual value Ch.2 <-> Data Pointer/CurrentActualValues[1]
//     Term 54 (AT2200-0500)/CC Inputs/Current actual value Ch.20 <-> Data Pointer/CurrentActualValues[19]
//     Term 54 (AT2200-0500)/CC Inputs/Current actual value Ch.21 <-> Data Pointer/CurrentActualValues[20]
//     Term 54 (AT2200-0500)/CC Inputs/Current actual value Ch.22 <-> Data Pointer/CurrentActualValues[21]
//     Term 54 (AT2200-0500)/CC Inputs/Current actual value Ch.23 <-> Data Pointer/CurrentActualValues[22]
//     Term 54 (AT2200-0500)/CC Inputs/Current actual value Ch.24 <-> Data Pointer/CurrentActualValues[23]
//     Term 54 (AT2200-0500)/CC Inputs/Current actual value Ch.25 <-> Data Pointer/CurrentActualValues[24]
//     Term 54 (AT2200-0500)/CC Inputs/Current actual value Ch.26 <-> Data Pointer/CurrentActualValues[25]
//     Term 54 (AT2200-0500)/CC Inputs/Current actual value Ch.27 <-> Data Pointer/CurrentActualValues[26]
//     Term 54 (AT2200-0500)/CC Inputs/Current actual value Ch.28 <-> Data Pointer/CurrentActualValues[27]
//     Term 54 (AT2200-0500)/CC Inputs/Current actual value Ch.29 <-> Data Pointer/CurrentActualValues[28]
//     Term 54 (AT2200-0500)/CC Inputs/Current actual value Ch.3 <-> Data Pointer/CurrentActualValues[2]
//     Term 54 (AT2200-0500)/CC Inputs/Current actual value Ch.30 <-> Data Pointer/CurrentActualValues[29]
//     Term 54 (AT2200-0500)/CC Inputs/Current actual value Ch.4 <-> Data Pointer/CurrentActualValues[3]
//     Term 54 (AT2200-0500)/CC Inputs/Current actual value Ch.5 <-> Data Pointer/CurrentActualValues[4]
//     Term 54 (AT2200-0500)/CC Inputs/Current actual value Ch.6 <-> Data Pointer/CurrentActualValues[5]
//     Term 54 (AT2200-0500)/CC Inputs/Current actual value Ch.7 <-> Data Pointer/CurrentActualValues[6]
//     Term 54 (AT2200-0500)/CC Inputs/Current actual value Ch.8 <-> Data Pointer/CurrentActualValues[7]
//     Term 54 (AT2200-0500)/CC Inputs/Current actual value Ch.9 <-> Data Pointer/CurrentActualValues[8]
//     Term 54 (AT2200-0500)/CC Inputs/Status <-> Data Pointer/Status
//     Term 54 (AT2200-0500)/CC Outputs/Control <-> Data Pointer/Control
//     Term 54 (AT2200-0500)/CC Outputs/Current setpoint value Ch.1 <-> Data Pointer/CurrentSetpointValues[0]
//     Term 54 (AT2200-0500)/CC Outputs/Current setpoint value Ch.10 <-> Data Pointer/CurrentSetpointValues[9]
//     Term 54 (AT2200-0500)/CC Outputs/Current setpoint value Ch.11 <-> Data Pointer/CurrentSetpointValues[10]
//     Term 54 (AT2200-0500)/CC Outputs/Current setpoint value Ch.12 <-> Data Pointer/CurrentSetpointValues[11]
//     Term 54 (AT2200-0500)/CC Outputs/Current setpoint value Ch.13 <-> Data Pointer/CurrentSetpointValues[12]
//     Term 54 (AT2200-0500)/CC Outputs/Current setpoint value Ch.14 <-> Data Pointer/CurrentSetpointValues[13]
//     Term 54 (AT2200-0500)/CC Outputs/Current setpoint value Ch.15 <-> Data Pointer/CurrentSetpointValues[14]
//     Term 54 (AT2200-0500)/CC Outputs/Current setpoint value Ch.16 <-> Data Pointer/CurrentSetpointValues[15]
//     Term 54 (AT2200-0500)/CC Outputs/Current setpoint value Ch.17 <-> Data Pointer/CurrentSetpointValues[16]
//     Term 54 (AT2200-0500)/CC Outputs/Current setpoint value Ch.18 <-> Data Pointer/CurrentSetpointValues[17]
//     Term 54 (AT2200-0500)/CC Outputs/Current setpoint value Ch.19 <-> Data Pointer/CurrentSetpointValues[18]
//     Term 54 (AT2200-0500)/CC Outputs/Current setpoint value Ch.2 <-> Data Pointer/CurrentSetpointValues[1]
//     Term 54 (AT2200-0500)/CC Outputs/Current setpoint value Ch.20 <-> Data Pointer/CurrentSetpointValues[19]
//     Term 54 (AT2200-0500)/CC Outputs/Current setpoint value Ch.21 <-> Data Pointer/CurrentSetpointValues[20]
//     Term 54 (AT2200-0500)/CC Outputs/Current setpoint value Ch.22 <-> Data Pointer/CurrentSetpointValues[21]
//     Term 54 (AT2200-0500)/CC Outputs/Current setpoint value Ch.23 <-> Data Pointer/CurrentSetpointValues[22]
//     Term 54 (AT2200-0500)/CC Outputs/Current setpoint value Ch.24 <-> Data Pointer/CurrentSetpointValues[23]
//     Term 54 (AT2200-0500)/CC Outputs/Current setpoint value Ch.25 <-> Data Pointer/CurrentSetpointValues[24]
//     Term 54 (AT2200-0500)/CC Outputs/Current setpoint value Ch.26 <-> Data Pointer/CurrentSetpointValues[25]
//     Term 54 (AT2200-0500)/CC Outputs/Current setpoint value Ch.27 <-> Data Pointer/CurrentSetpointValues[26]
//     Term 54 (AT2200-0500)/CC Outputs/Current setpoint value Ch.28 <-> Data Pointer/CurrentSetpointValues[27]
//     Term 54 (AT2200-0500)/CC Outputs/Current setpoint value Ch.29 <-> Data Pointer/CurrentSetpointValues[28]
//     Term 54 (AT2200-0500)/CC Outputs/Current setpoint value Ch.3 <-> Data Pointer/CurrentSetpointValues[2]
//     Term 54 (AT2200-0500)/CC Outputs/Current setpoint value Ch.30 <-> Data Pointer/CurrentSetpointValues[29]
//     Term 54 (AT2200-0500)/CC Outputs/Current setpoint value Ch.4 <-> Data Pointer/CurrentSetpointValues[3]
//     Term 54 (AT2200-0500)/CC Outputs/Current setpoint value Ch.5 <-> Data Pointer/CurrentSetpointValues[4]
//     Term 54 (AT2200-0500)/CC Outputs/Current setpoint value Ch.6 <-> Data Pointer/CurrentSetpointValues[5]
//     Term 54 (AT2200-0500)/CC Outputs/Current setpoint value Ch.7 <-> Data Pointer/CurrentSetpointValues[6]
//     Term 54 (AT2200-0500)/CC Outputs/Current setpoint value Ch.8 <-> Data Pointer/CurrentSetpointValues[7]
//     Term 54 (AT2200-0500)/CC Outputs/Current setpoint value Ch.9 <-> Data Pointer/CurrentSetpointValues[8]
//     Term 54 (AT2200-0500)/LFB Inputs/BinaryData <-> Data Pointer/HallSensorValues
//   Device 29 <-> TcCOM Objects/XTS ProcessingUnit 1/Part 1/Module 43
//     Term 55 (AT2000-0250)/CC Inputs/Current actual value Ch.1 <-> Data Pointer/CurrentActualValues[0]
//     Term 55 (AT2000-0250)/CC Inputs/Current actual value Ch.10 <-> Data Pointer/CurrentActualValues[9]
//     Term 55 (AT2000-0250)/CC Inputs/Current actual value Ch.11 <-> Data Pointer/CurrentActualValues[10]
//     Term 55 (AT2000-0250)/CC Inputs/Current actual value Ch.12 <-> Data Pointer/CurrentActualValues[11]
//     Term 55 (AT2000-0250)/CC Inputs/Current actual value Ch.13 <-> Data Pointer/CurrentActualValues[12]
//     Term 55 (AT2000-0250)/CC Inputs/Current actual value Ch.14 <-> Data Pointer/CurrentActualValues[13]
//     Term 55 (AT2000-0250)/CC Inputs/Current actual value Ch.15 <-> Data Pointer/CurrentActualValues[14]
//     Term 55 (AT2000-0250)/CC Inputs/Current actual value Ch.2 <-> Data Pointer/CurrentActualValues[1]
//     Term 55 (AT2000-0250)/CC Inputs/Current actual value Ch.3 <-> Data Pointer/CurrentActualValues[2]
//     Term 55 (AT2000-0250)/CC Inputs/Current actual value Ch.4 <-> Data Pointer/CurrentActualValues[3]
//     Term 55 (AT2000-0250)/CC Inputs/Current actual value Ch.5 <-> Data Pointer/CurrentActualValues[4]
//     Term 55 (AT2000-0250)/CC Inputs/Current actual value Ch.6 <-> Data Pointer/CurrentActualValues[5]
//     Term 55 (AT2000-0250)/CC Inputs/Current actual value Ch.7 <-> Data Pointer/CurrentActualValues[6]
//     Term 55 (AT2000-0250)/CC Inputs/Current actual value Ch.8 <-> Data Pointer/CurrentActualValues[7]
//     Term 55 (AT2000-0250)/CC Inputs/Current actual value Ch.9 <-> Data Pointer/CurrentActualValues[8]
//     Term 55 (AT2000-0250)/CC Inputs/Status <-> Data Pointer/Status
//     Term 55 (AT2000-0250)/CC Outputs/Control <-> Data Pointer/Control
//     Term 55 (AT2000-0250)/CC Outputs/Current setpoint value Ch.1 <-> Data Pointer/CurrentSetpointValues[0]
//     Term 55 (AT2000-0250)/CC Outputs/Current setpoint value Ch.10 <-> Data Pointer/CurrentSetpointValues[9]
//     Term 55 (AT2000-0250)/CC Outputs/Current setpoint value Ch.11 <-> Data Pointer/CurrentSetpointValues[10]
//     Term 55 (AT2000-0250)/CC Outputs/Current setpoint value Ch.12 <-> Data Pointer/CurrentSetpointValues[11]
//     Term 55 (AT2000-0250)/CC Outputs/Current setpoint value Ch.13 <-> Data Pointer/CurrentSetpointValues[12]
//     Term 55 (AT2000-0250)/CC Outputs/Current setpoint value Ch.14 <-> Data Pointer/CurrentSetpointValues[13]
//     Term 55 (AT2000-0250)/CC Outputs/Current setpoint value Ch.15 <-> Data Pointer/CurrentSetpointValues[14]
//     Term 55 (AT2000-0250)/CC Outputs/Current setpoint value Ch.2 <-> Data Pointer/CurrentSetpointValues[1]
//     Term 55 (AT2000-0250)/CC Outputs/Current setpoint value Ch.3 <-> Data Pointer/CurrentSetpointValues[2]
//     Term 55 (AT2000-0250)/CC Outputs/Current setpoint value Ch.4 <-> Data Pointer/CurrentSetpointValues[3]
//     Term 55 (AT2000-0250)/CC Outputs/Current setpoint value Ch.5 <-> Data Pointer/CurrentSetpointValues[4]
//     Term 55 (AT2000-0250)/CC Outputs/Current setpoint value Ch.6 <-> Data Pointer/CurrentSetpointValues[5]
//     Term 55 (AT2000-0250)/CC Outputs/Current setpoint value Ch.7 <-> Data Pointer/CurrentSetpointValues[6]
//     Term 55 (AT2000-0250)/CC Outputs/Current setpoint value Ch.8 <-> Data Pointer/CurrentSetpointValues[7]
//     Term 55 (AT2000-0250)/CC Outputs/Current setpoint value Ch.9 <-> Data Pointer/CurrentSetpointValues[8]
//     Term 55 (AT2000-0250)/Term 56 (AT2000-5250)/FB Inputs/Value Channel 01 <-> Data Pointer/RawPositionValues[0]
//     Term 55 (AT2000-0250)/Term 56 (AT2000-5250)/FB Inputs/Value Channel 02 <-> Data Pointer/RawPositionValues[1]
//     Term 55 (AT2000-0250)/Term 56 (AT2000-5250)/FB Inputs/Value Channel 03 <-> Data Pointer/RawPositionValues[2]
//     Term 55 (AT2000-0250)/Term 56 (AT2000-5250)/FB Inputs/Value Channel 04 <-> Data Pointer/RawPositionValues[3]
//     Term 55 (AT2000-0250)/Term 56 (AT2000-5250)/FB Inputs/Value Channel 05 <-> Data Pointer/RawPositionValues[4]
//     Term 55 (AT2000-0250)/Term 56 (AT2000-5250)/FB Inputs/Value Channel 06 <-> Data Pointer/RawPositionValues[5]
//     Term 55 (AT2000-0250)/Term 56 (AT2000-5250)/FB Inputs/Value Channel 07 <-> Data Pointer/RawPositionValues[6]
//     Term 55 (AT2000-0250)/Term 56 (AT2000-5250)/FB Inputs/Value Channel 08 <-> Data Pointer/RawPositionValues[7]
//     Term 55 (AT2000-0250)/Term 56 (AT2000-5250)/FB Inputs/Value Channel 09 <-> Data Pointer/RawPositionValues[8]
//     Term 55 (AT2000-0250)/Term 56 (AT2000-5250)/FB Inputs/Value Channel 10 <-> Data Pointer/RawPositionValues[9]
//     Term 55 (AT2000-0250)/Term 56 (AT2000-5250)/FB Inputs/Value Channel 11 <-> Data Pointer/RawPositionValues[10]
//     Term 55 (AT2000-0250)/Term 56 (AT2000-5250)/FB Inputs/Value Channel 12 <-> Data Pointer/RawPositionValues[11]
//     Term 55 (AT2000-0250)/Term 56 (AT2000-5250)/FB Inputs/Value Channel 13 <-> Data Pointer/RawPositionValues[12]
//     Term 55 (AT2000-0250)/Term 56 (AT2000-5250)/FB Inputs/Value Channel 14 <-> Data Pointer/RawPositionValues[13]
//     Term 55 (AT2000-0250)/Term 56 (AT2000-5250)/FB Inputs/Value Channel 15 <-> Data Pointer/RawPositionValues[14]
//     Term 55 (AT2000-0250)/Term 56 (AT2000-5250)/FB Inputs/Value Channel 16 <-> Data Pointer/RawPositionValues[15]
//     Term 55 (AT2000-0250)/Term 56 (AT2000-5250)/FB Inputs/Value Channel 17 <-> Data Pointer/RawPositionValues[16]
//     Term 55 (AT2000-0250)/Term 56 (AT2000-5250)/FB Inputs/Value Channel 18 <-> Data Pointer/RawPositionValues[17]
//     Term 55 (AT2000-0250)/Term 56 (AT2000-5250)/FB Inputs/Value Channel 19 <-> Data Pointer/RawPositionValues[18]
//     Term 55 (AT2000-0250)/Term 56 (AT2000-5250)/FB Inputs/Value Channel 20 <-> Data Pointer/RawPositionValues[19]
//     Term 55 (AT2000-0250)/Term 56 (AT2000-5250)/FB Inputs/Value Channel 21 <-> Data Pointer/RawPositionValues[20]
//     Term 55 (AT2000-0250)/Term 56 (AT2000-5250)/FB Inputs/Value Channel 22 <-> Data Pointer/RawPositionValues[21]
//     Term 55 (AT2000-0250)/Term 56 (AT2000-5250)/FB Inputs/Value Channel 23 <-> Data Pointer/RawPositionValues[22]
//     Term 55 (AT2000-0250)/Term 56 (AT2000-5250)/FB Inputs/Value Channel 24 <-> Data Pointer/RawPositionValues[23]
//     Term 55 (AT2000-0250)/Term 56 (AT2000-5250)/FB Inputs/Value Channel 25 <-> Data Pointer/RawPositionValues[24]
//     Term 55 (AT2000-0250)/Term 56 (AT2000-5250)/FB Inputs/Value Channel 26 <-> Data Pointer/RawPositionValues[25]
//     Term 55 (AT2000-0250)/Term 56 (AT2000-5250)/FB Inputs/Value Channel 27 <-> Data Pointer/RawPositionValues[26]
//     Term 55 (AT2000-0250)/Term 56 (AT2000-5250)/FB Inputs/Value Channel 28 <-> Data Pointer/RawPositionValues[27]
//     Term 55 (AT2000-0250)/Term 56 (AT2000-5250)/FB Inputs/Value Channel 29 <-> Data Pointer/RawPositionValues[28]
//     Term 55 (AT2000-0250)/Term 56 (AT2000-5250)/FB Inputs/Value Channel 30 <-> Data Pointer/RawPositionValues[29]
//     Term 55 (AT2000-0250)/Term 56 (AT2000-5250)/FB Inputs/Value Channel 31 <-> Data Pointer/RawPositionValues[30]
//     Term 55 (AT2000-0250)/Term 56 (AT2000-5250)/FB Inputs/Value Channel 32 <-> Data Pointer/RawPositionValues[31]
//   Device 30 <-> TcCOM Objects/XTS ProcessingUnit 1/Part 1/Module 44
//     Term 57 (AT2002-0250)/CC Inputs/Current actual value Ch.1 <-> Data Pointer/CurrentActualValues[0]
//     Term 57 (AT2002-0250)/CC Inputs/Current actual value Ch.10 <-> Data Pointer/CurrentActualValues[9]
//     Term 57 (AT2002-0250)/CC Inputs/Current actual value Ch.11 <-> Data Pointer/CurrentActualValues[10]
//     Term 57 (AT2002-0250)/CC Inputs/Current actual value Ch.12 <-> Data Pointer/CurrentActualValues[11]
//     Term 57 (AT2002-0250)/CC Inputs/Current actual value Ch.13 <-> Data Pointer/CurrentActualValues[12]
//     Term 57 (AT2002-0250)/CC Inputs/Current actual value Ch.14 <-> Data Pointer/CurrentActualValues[13]
//     Term 57 (AT2002-0250)/CC Inputs/Current actual value Ch.15 <-> Data Pointer/CurrentActualValues[14]
//     Term 57 (AT2002-0250)/CC Inputs/Current actual value Ch.2 <-> Data Pointer/CurrentActualValues[1]
//     Term 57 (AT2002-0250)/CC Inputs/Current actual value Ch.3 <-> Data Pointer/CurrentActualValues[2]
//     Term 57 (AT2002-0250)/CC Inputs/Current actual value Ch.4 <-> Data Pointer/CurrentActualValues[3]
//     Term 57 (AT2002-0250)/CC Inputs/Current actual value Ch.5 <-> Data Pointer/CurrentActualValues[4]
//     Term 57 (AT2002-0250)/CC Inputs/Current actual value Ch.6 <-> Data Pointer/CurrentActualValues[5]
//     Term 57 (AT2002-0250)/CC Inputs/Current actual value Ch.7 <-> Data Pointer/CurrentActualValues[6]
//     Term 57 (AT2002-0250)/CC Inputs/Current actual value Ch.8 <-> Data Pointer/CurrentActualValues[7]
//     Term 57 (AT2002-0250)/CC Inputs/Current actual value Ch.9 <-> Data Pointer/CurrentActualValues[8]
//     Term 57 (AT2002-0250)/CC Inputs/Status <-> Data Pointer/Status
//     Term 57 (AT2002-0250)/CC Outputs/Control <-> Data Pointer/Control
//     Term 57 (AT2002-0250)/CC Outputs/Current setpoint value Ch.1 <-> Data Pointer/CurrentSetpointValues[0]
//     Term 57 (AT2002-0250)/CC Outputs/Current setpoint value Ch.10 <-> Data Pointer/CurrentSetpointValues[9]
//     Term 57 (AT2002-0250)/CC Outputs/Current setpoint value Ch.11 <-> Data Pointer/CurrentSetpointValues[10]
//     Term 57 (AT2002-0250)/CC Outputs/Current setpoint value Ch.12 <-> Data Pointer/CurrentSetpointValues[11]
//     Term 57 (AT2002-0250)/CC Outputs/Current setpoint value Ch.13 <-> Data Pointer/CurrentSetpointValues[12]
//     Term 57 (AT2002-0250)/CC Outputs/Current setpoint value Ch.14 <-> Data Pointer/CurrentSetpointValues[13]
//     Term 57 (AT2002-0250)/CC Outputs/Current setpoint value Ch.15 <-> Data Pointer/CurrentSetpointValues[14]
//     Term 57 (AT2002-0250)/CC Outputs/Current setpoint value Ch.2 <-> Data Pointer/CurrentSetpointValues[1]
//     Term 57 (AT2002-0250)/CC Outputs/Current setpoint value Ch.3 <-> Data Pointer/CurrentSetpointValues[2]
//     Term 57 (AT2002-0250)/CC Outputs/Current setpoint value Ch.4 <-> Data Pointer/CurrentSetpointValues[3]
//     Term 57 (AT2002-0250)/CC Outputs/Current setpoint value Ch.5 <-> Data Pointer/CurrentSetpointValues[4]
//     Term 57 (AT2002-0250)/CC Outputs/Current setpoint value Ch.6 <-> Data Pointer/CurrentSetpointValues[5]
//     Term 57 (AT2002-0250)/CC Outputs/Current setpoint value Ch.7 <-> Data Pointer/CurrentSetpointValues[6]
//     Term 57 (AT2002-0250)/CC Outputs/Current setpoint value Ch.8 <-> Data Pointer/CurrentSetpointValues[7]
//     Term 57 (AT2002-0250)/CC Outputs/Current setpoint value Ch.9 <-> Data Pointer/CurrentSetpointValues[8]
//     Term 57 (AT2002-0250)/Term 58 (AT2002-5250)/FB Inputs/Value Channel 01 <-> Data Pointer/RawPositionValues[0]
//     Term 57 (AT2002-0250)/Term 58 (AT2002-5250)/FB Inputs/Value Channel 02 <-> Data Pointer/RawPositionValues[1]
//     Term 57 (AT2002-0250)/Term 58 (AT2002-5250)/FB Inputs/Value Channel 03 <-> Data Pointer/RawPositionValues[2]
//     Term 57 (AT2002-0250)/Term 58 (AT2002-5250)/FB Inputs/Value Channel 04 <-> Data Pointer/RawPositionValues[3]
//     Term 57 (AT2002-0250)/Term 58 (AT2002-5250)/FB Inputs/Value Channel 05 <-> Data Pointer/RawPositionValues[4]
//     Term 57 (AT2002-0250)/Term 58 (AT2002-5250)/FB Inputs/Value Channel 06 <-> Data Pointer/RawPositionValues[5]
//     Term 57 (AT2002-0250)/Term 58 (AT2002-5250)/FB Inputs/Value Channel 07 <-> Data Pointer/RawPositionValues[6]
//     Term 57 (AT2002-0250)/Term 58 (AT2002-5250)/FB Inputs/Value Channel 08 <-> Data Pointer/RawPositionValues[7]
//     Term 57 (AT2002-0250)/Term 58 (AT2002-5250)/FB Inputs/Value Channel 09 <-> Data Pointer/RawPositionValues[8]
//     Term 57 (AT2002-0250)/Term 58 (AT2002-5250)/FB Inputs/Value Channel 10 <-> Data Pointer/RawPositionValues[9]
//     Term 57 (AT2002-0250)/Term 58 (AT2002-5250)/FB Inputs/Value Channel 11 <-> Data Pointer/RawPositionValues[10]
//     Term 57 (AT2002-0250)/Term 58 (AT2002-5250)/FB Inputs/Value Channel 12 <-> Data Pointer/RawPositionValues[11]
//     Term 57 (AT2002-0250)/Term 58 (AT2002-5250)/FB Inputs/Value Channel 13 <-> Data Pointer/RawPositionValues[12]
